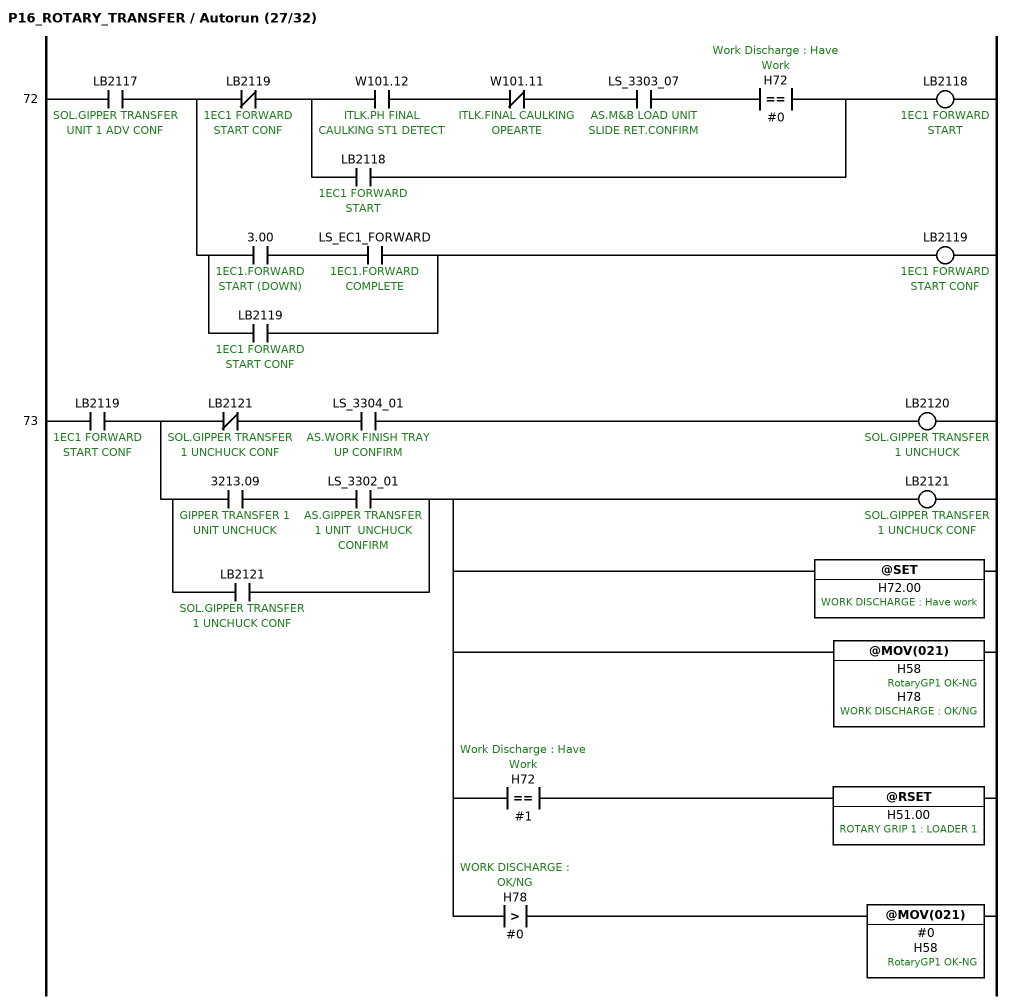
; [picture p264: P16_ROTARY_TRANSFER / Autorun, rungs 72-73]
; rung 72
LD LB2117  ; SOL.GIPPER TRANSFER UNIT 1 ADV CONF
OUT TR0
ANDNOT LB2119  ; 1EC1 FORWARD START CONF
LD W101.12  ; ITLK.PH FINAL CAULKING ST1 DETECT
ANDNOT W101.11  ; ITLK.FINAL CAULKING OPEARTE
AND LS_3303_07  ; AS.M&B LOAD UNIT SLIDE RET.CONFIRM
AND=(300) H72 #0  ; Work Discharge : Have Work
OR LB2118  ; 1EC1 FORWARD START
ANDLD
OUT LB2118  ; 1EC1 FORWARD START
LD TR0
LD 3.00  ; 1EC1.FORWARD START (DOWN)
AND LS_EC1_FORWARD  ; 1EC1.FORWARD COMPLETE
OR LB2119  ; 1EC1 FORWARD START CONF
ANDLD
OUT LB2119  ; 1EC1 FORWARD START CONF
; rung 73
LD LB2119  ; 1EC1 FORWARD START CONF
OUT TR0
ANDNOT LB2121  ; SOL.GIPPER TRANSFER 1 UNCHUCK CONF
AND LS_3304_01  ; AS.WORK FINISH TRAY UP CONFIRM
OUT LB2120  ; SOL.GIPPER TRANSFER 1 UNCHUCK
LD TR0
LD 3213.09  ; GIPPER TRANSFER 1 UNIT UNCHUCK
AND LS_3302_01  ; AS.GIPPER TRANSFER 1 UNIT  UNCHUCK CONFIRM
OR LB2121  ; SOL.GIPPER TRANSFER 1 UNCHUCK CONF
ANDLD
OUT TR0
OUT LB2121  ; SOL.GIPPER TRANSFER 1 UNCHUCK CONF
@SET H72.00  ; WORK DISCHARGE : Have work
@MOV(021) H58 H78  ; RotaryGP1 OK-NG, WORK DISCHARGE : OK/NG
AND=(300) H72 #1  ; Work Discharge : Have Work
@RSET H51.00  ; ROTARY GRIP 1 : LOADER 1
LD TR0
AND>(320) H78 #0  ; WORK DISCHARGE : OK/NG
@MOV(021) #0 H58  ; RotaryGP1 OK-NG

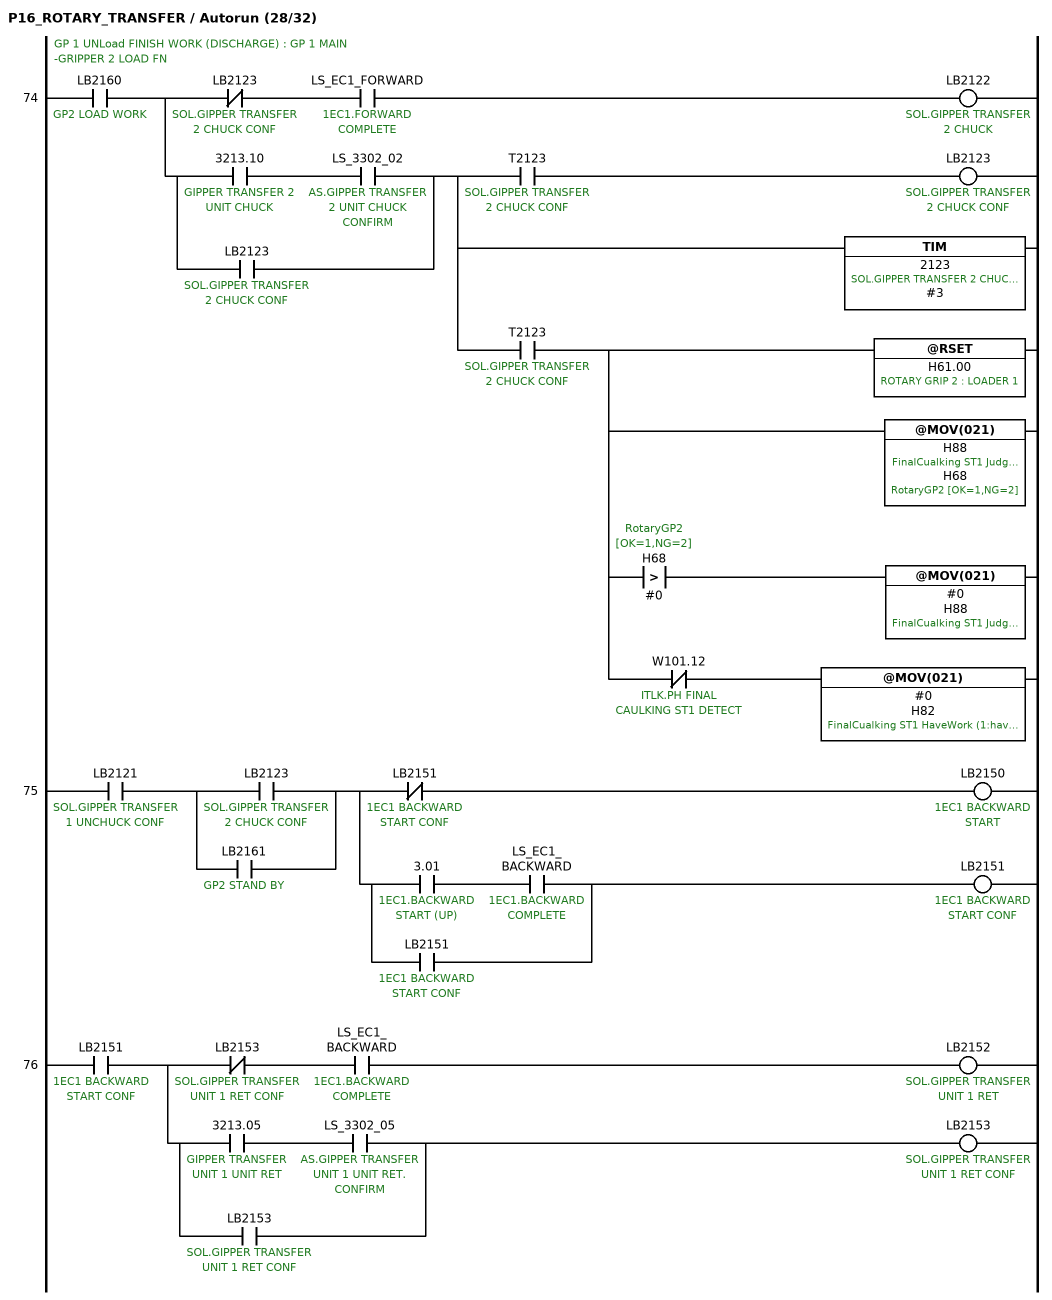
; rung 74: GP 1 UNLoad FINISH WORK (DISCHARGE) : GP 1 MAIN / -GRIPPER 2 LOAD FN
LD LB2160  ; GP2 LOAD WORK
OUT TR0
ANDNOT LB2123  ; SOL.GIPPER TRANSFER 2 CHUCK CONF
AND LS_EC1_FORWARD  ; 1EC1.FORWARD COMPLETE
OUT LB2122  ; SOL.GIPPER TRANSFER 2 CHUCK
LD TR0
LD 3213.10  ; GIPPER TRANSFER 2 UNIT CHUCK
AND LS_3302_02  ; AS.GIPPER TRANSFER 2 UNIT CHUCK CONFIRM
OR LB2123  ; SOL.GIPPER TRANSFER 2 CHUCK CONF
ANDLD
OUT TR0
AND T2123  ; SOL.GIPPER TRANSFER 2 CHUCK CONF
OUT LB2123  ; SOL.GIPPER TRANSFER 2 CHUCK CONF
LD TR0
TIM 2123 #3  ; SOL.GIPPER TRANSFER 2 CHUCK CONF
AND T2123  ; SOL.GIPPER TRANSFER 2 CHUCK CONF
OUT TR0
@RSET H61.00  ; ROTARY GRIP 2 : LOADER 1
@MOV(021) H88 H68  ; FinalCualking ST1 Judge [OK=1,NG=2], RotaryGP2 [OK=1,NG=2]
AND>(320) H68 #0  ; RotaryGP2 [OK=1,NG=2]
@MOV(021) #0 H88  ; FinalCualking ST1 Judge [OK=1,NG=2]
LD TR0
ANDNOT W101.12  ; ITLK.PH FINAL CAULKING ST1 DETECT
@MOV(021) #0 H82  ; FinalCualking ST1 HaveWork (1:have work 2:no work)
; rung 75
LD LB2121  ; SOL.GIPPER TRANSFER 1 UNCHUCK CONF
LD LB2123  ; SOL.GIPPER TRANSFER 2 CHUCK CONF
OR LB2161  ; GP2 STAND BY
ANDLD
OUT TR0
ANDNOT LB2151  ; 1EC1 BACKWARD START CONF
OUT LB2150  ; 1EC1 BACKWARD START
LD TR0
LD 3.01  ; 1EC1.BACKWARD START (UP)
AND LS_EC1_BACKWARD  ; 1EC1.BACKWARD COMPLETE
OR LB2151  ; 1EC1 BACKWARD START CONF
ANDLD
OUT LB2151  ; 1EC1 BACKWARD START CONF
; rung 76
LD LB2151  ; 1EC1 BACKWARD START CONF
OUT TR0
ANDNOT LB2153  ; SOL.GIPPER TRANSFER UNIT 1 RET CONF
AND LS_EC1_BACKWARD  ; 1EC1.BACKWARD COMPLETE
OUT LB2152  ; SOL.GIPPER TRANSFER UNIT 1 RET
LD TR0
LD 3213.05  ; GIPPER TRANSFER UNIT 1 UNIT RET
AND LS_3302_05  ; AS.GIPPER TRANSFER UNIT 1 UNIT RET. CONFIRM
OR LB2153  ; SOL.GIPPER TRANSFER UNIT 1 RET CONF
ANDLD
OUT LB2153  ; SOL.GIPPER TRANSFER UNIT 1 RET CONF

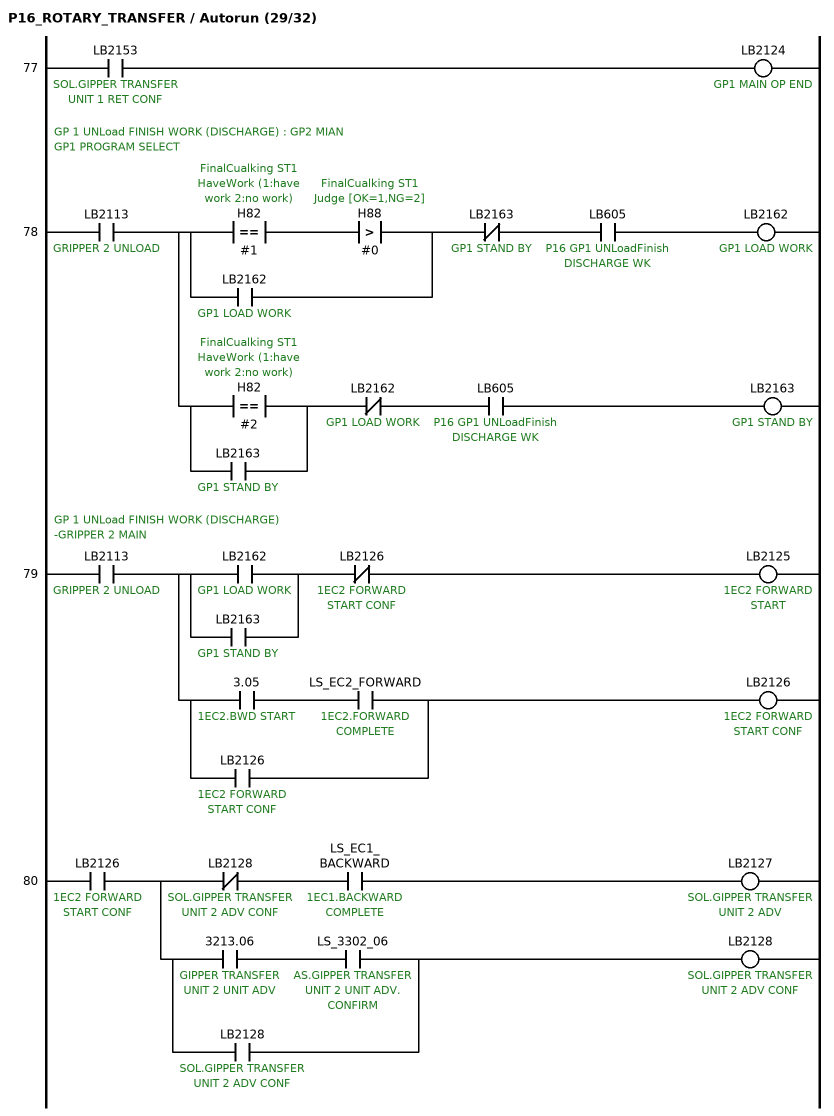
; rung 77
LD LB2153  ; SOL.GIPPER TRANSFER UNIT 1 RET CONF
OUT LB2124  ; GP1 MAIN OP END
; rung 78: GP 1 UNLoad FINISH WORK (DISCHARGE) : GP2 MIAN / GP1 PROGRAM SELECT
LD LB2113  ; GRIPPER 2 UNLOAD
OUT TR0
LD=(300) H82 #1  ; FinalCualking ST1 HaveWork (1:have work 2:no work)
AND>(320) H88 #0  ; FinalCualking ST1 Judge [OK=1,NG=2]
OR LB2162  ; GP1 LOAD WORK
ANDLD
ANDNOT LB2163  ; GP1 STAND BY
AND LB605  ; P16 GP1 UNLoadFinish DISCHARGE WK
OUT LB2162  ; GP1 LOAD WORK
LD TR0
LD=(300) H82 #2  ; FinalCualking ST1 HaveWork (1:have work 2:no work)
OR LB2163  ; GP1 STAND BY
ANDLD
ANDNOT LB2162  ; GP1 LOAD WORK
AND LB605  ; P16 GP1 UNLoadFinish DISCHARGE WK
OUT LB2163  ; GP1 STAND BY
; rung 79: GP 1 UNLoad FINISH WORK (DISCHARGE) / -GRIPPER 2 MAIN
LD LB2113  ; GRIPPER 2 UNLOAD
OUT TR0
LD LB2162  ; GP1 LOAD WORK
OR LB2163  ; GP1 STAND BY
ANDLD
ANDNOT LB2126  ; 1EC2 FORWARD START CONF
OUT LB2125  ; 1EC2 FORWARD START
LD TR0
LD 3.05  ; 1EC2.BWD START
AND LS_EC2_FORWARD  ; 1EC2.FORWARD COMPLETE
OR LB2126  ; 1EC2 FORWARD START CONF
ANDLD
OUT LB2126  ; 1EC2 FORWARD START CONF
; rung 80
LD LB2126  ; 1EC2 FORWARD START CONF
OUT TR0
ANDNOT LB2128  ; SOL.GIPPER TRANSFER UNIT 2 ADV CONF
AND LS_EC1_BACKWARD  ; 1EC1.BACKWARD COMPLETE
OUT LB2127  ; SOL.GIPPER TRANSFER UNIT 2 ADV
LD TR0
LD 3213.06  ; GIPPER TRANSFER UNIT 2 UNIT ADV
AND LS_3302_06  ; AS.GIPPER TRANSFER UNIT 2 UNIT ADV. CONFIRM
OR LB2128  ; SOL.GIPPER TRANSFER UNIT 2 ADV CONF
ANDLD
OUT LB2128  ; SOL.GIPPER TRANSFER UNIT 2 ADV CONF

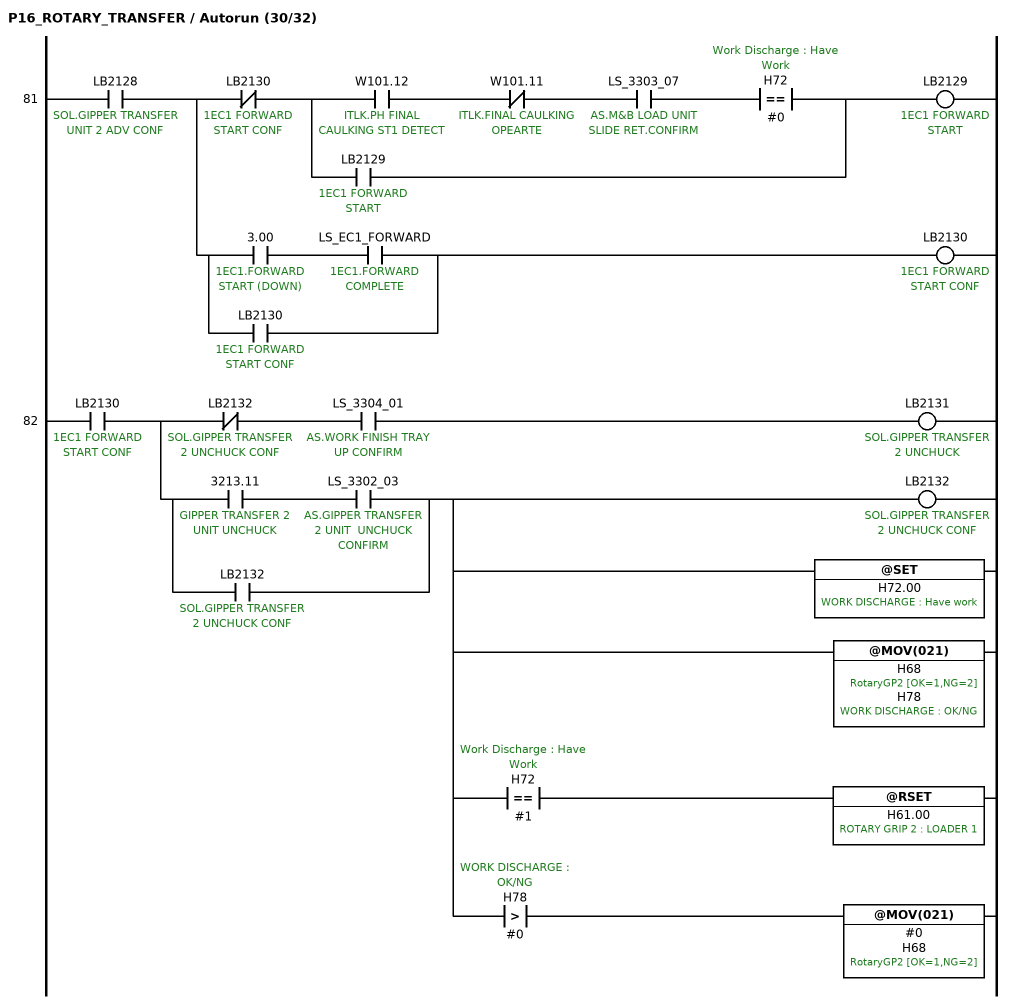
; rung 81
LD LB2128  ; SOL.GIPPER TRANSFER UNIT 2 ADV CONF
OUT TR0
ANDNOT LB2130  ; 1EC1 FORWARD START CONF
LD W101.12  ; ITLK.PH FINAL CAULKING ST1 DETECT
ANDNOT W101.11  ; ITLK.FINAL CAULKING OPEARTE
AND LS_3303_07  ; AS.M&B LOAD UNIT SLIDE RET.CONFIRM
AND=(300) H72 #0  ; Work Discharge : Have Work
OR LB2129  ; 1EC1 FORWARD START
ANDLD
OUT LB2129  ; 1EC1 FORWARD START
LD TR0
LD 3.00  ; 1EC1.FORWARD START (DOWN)
AND LS_EC1_FORWARD  ; 1EC1.FORWARD COMPLETE
OR LB2130  ; 1EC1 FORWARD START CONF
ANDLD
OUT LB2130  ; 1EC1 FORWARD START CONF
; rung 82
LD LB2130  ; 1EC1 FORWARD START CONF
OUT TR0
ANDNOT LB2132  ; SOL.GIPPER TRANSFER 2 UNCHUCK CONF
AND LS_3304_01  ; AS.WORK FINISH TRAY UP CONFIRM
OUT LB2131  ; SOL.GIPPER TRANSFER 2 UNCHUCK
LD TR0
LD 3213.11  ; GIPPER TRANSFER 2 UNIT UNCHUCK
AND LS_3302_03  ; AS.GIPPER TRANSFER 2 UNIT  UNCHUCK CONFIRM
OR LB2132  ; SOL.GIPPER TRANSFER 2 UNCHUCK CONF
ANDLD
OUT TR0
OUT LB2132  ; SOL.GIPPER TRANSFER 2 UNCHUCK CONF
@SET H72.00  ; WORK DISCHARGE : Have work
@MOV(021) H68 H78  ; RotaryGP2 [OK=1,NG=2], WORK DISCHARGE : OK/NG
AND=(300) H72 #1  ; Work Discharge : Have Work
@RSET H61.00  ; ROTARY GRIP 2 : LOADER 1
LD TR0
AND>(320) H78 #0  ; WORK DISCHARGE : OK/NG
@MOV(021) #0 H68  ; RotaryGP2 [OK=1,NG=2]

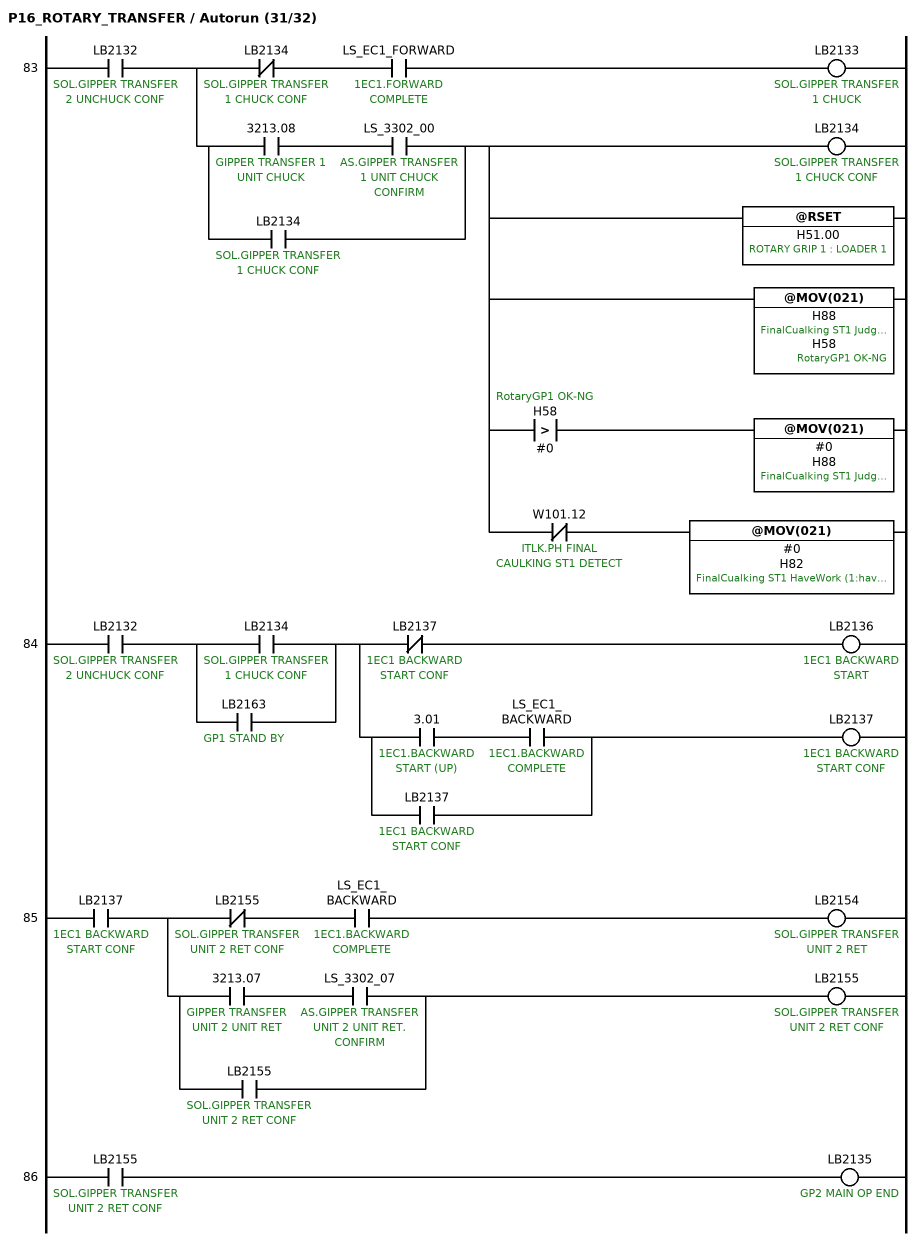
; rung 83
LD LB2132  ; SOL.GIPPER TRANSFER 2 UNCHUCK CONF
OUT TR0
ANDNOT LB2134  ; SOL.GIPPER TRANSFER 1 CHUCK CONF
AND LS_EC1_FORWARD  ; 1EC1.FORWARD COMPLETE
OUT LB2133  ; SOL.GIPPER TRANSFER 1 CHUCK
LD TR0
LD 3213.08  ; GIPPER TRANSFER 1 UNIT CHUCK
AND LS_3302_00  ; AS.GIPPER TRANSFER 1 UNIT CHUCK CONFIRM
OR LB2134  ; SOL.GIPPER TRANSFER 1 CHUCK CONF
ANDLD
OUT TR0
OUT LB2134  ; SOL.GIPPER TRANSFER 1 CHUCK CONF
@RSET H51.00  ; ROTARY GRIP 1 : LOADER 1
@MOV(021) H88 H58  ; FinalCualking ST1 Judge [OK=1,NG=2], RotaryGP1 OK-NG
AND>(320) H58 #0  ; RotaryGP1 OK-NG
@MOV(021) #0 H88  ; FinalCualking ST1 Judge [OK=1,NG=2]
LD TR0
ANDNOT W101.12  ; ITLK.PH FINAL CAULKING ST1 DETECT
@MOV(021) #0 H82  ; FinalCualking ST1 HaveWork (1:have work 2:no work)
; rung 84
LD LB2132  ; SOL.GIPPER TRANSFER 2 UNCHUCK CONF
LD LB2134  ; SOL.GIPPER TRANSFER 1 CHUCK CONF
OR LB2163  ; GP1 STAND BY
ANDLD
OUT TR0
ANDNOT LB2137  ; 1EC1 BACKWARD START CONF
OUT LB2136  ; 1EC1 BACKWARD START
LD TR0
LD 3.01  ; 1EC1.BACKWARD START (UP)
AND LS_EC1_BACKWARD  ; 1EC1.BACKWARD COMPLETE
OR LB2137  ; 1EC1 BACKWARD START CONF
ANDLD
OUT LB2137  ; 1EC1 BACKWARD START CONF
; rung 85
LD LB2137  ; 1EC1 BACKWARD START CONF
OUT TR0
ANDNOT LB2155  ; SOL.GIPPER TRANSFER UNIT 2 RET CONF
AND LS_EC1_BACKWARD  ; 1EC1.BACKWARD COMPLETE
OUT LB2154  ; SOL.GIPPER TRANSFER UNIT 2 RET
LD TR0
LD 3213.07  ; GIPPER TRANSFER UNIT 2 UNIT RET
AND LS_3302_07  ; AS.GIPPER TRANSFER UNIT 2 UNIT RET. CONFIRM
OR LB2155  ; SOL.GIPPER TRANSFER UNIT 2 RET CONF
ANDLD
OUT LB2155  ; SOL.GIPPER TRANSFER UNIT 2 RET CONF
; rung 86
LD LB2155  ; SOL.GIPPER TRANSFER UNIT 2 RET CONF
OUT LB2135  ; GP2 MAIN OP END

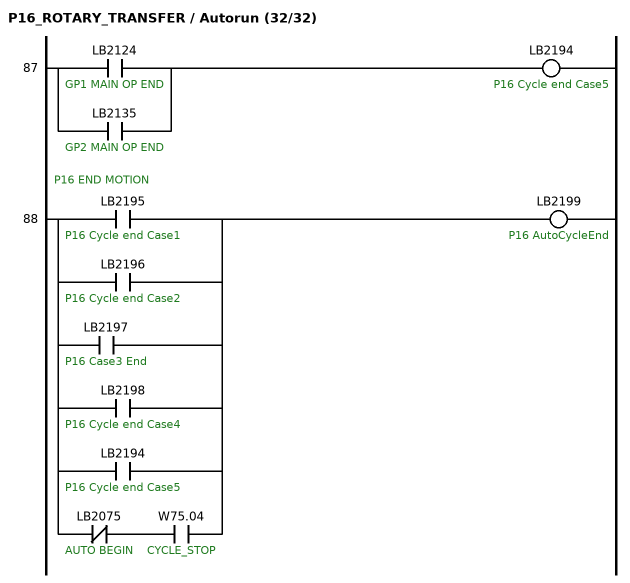
; rung 87
LD LB2124  ; GP1 MAIN OP END
OR LB2135  ; GP2 MAIN OP END
OUT LB2194  ; P16 Cycle end Case5
; rung 88: P16 END MOTION
LD LB2195  ; P16 Cycle end Case1
OR LB2196  ; P16 Cycle end Case2
OR LB2197  ; P16 Case3 End
OR LB2198  ; P16 Cycle end Case4
OR LB2194  ; P16 Cycle end Case5
LDNOT LB2075  ; AUTO BEGIN
AND W75.04  ; CYCLE_STOP
ORLD
OUT LB2199  ; P16 AutoCycleEnd

### Section Condition

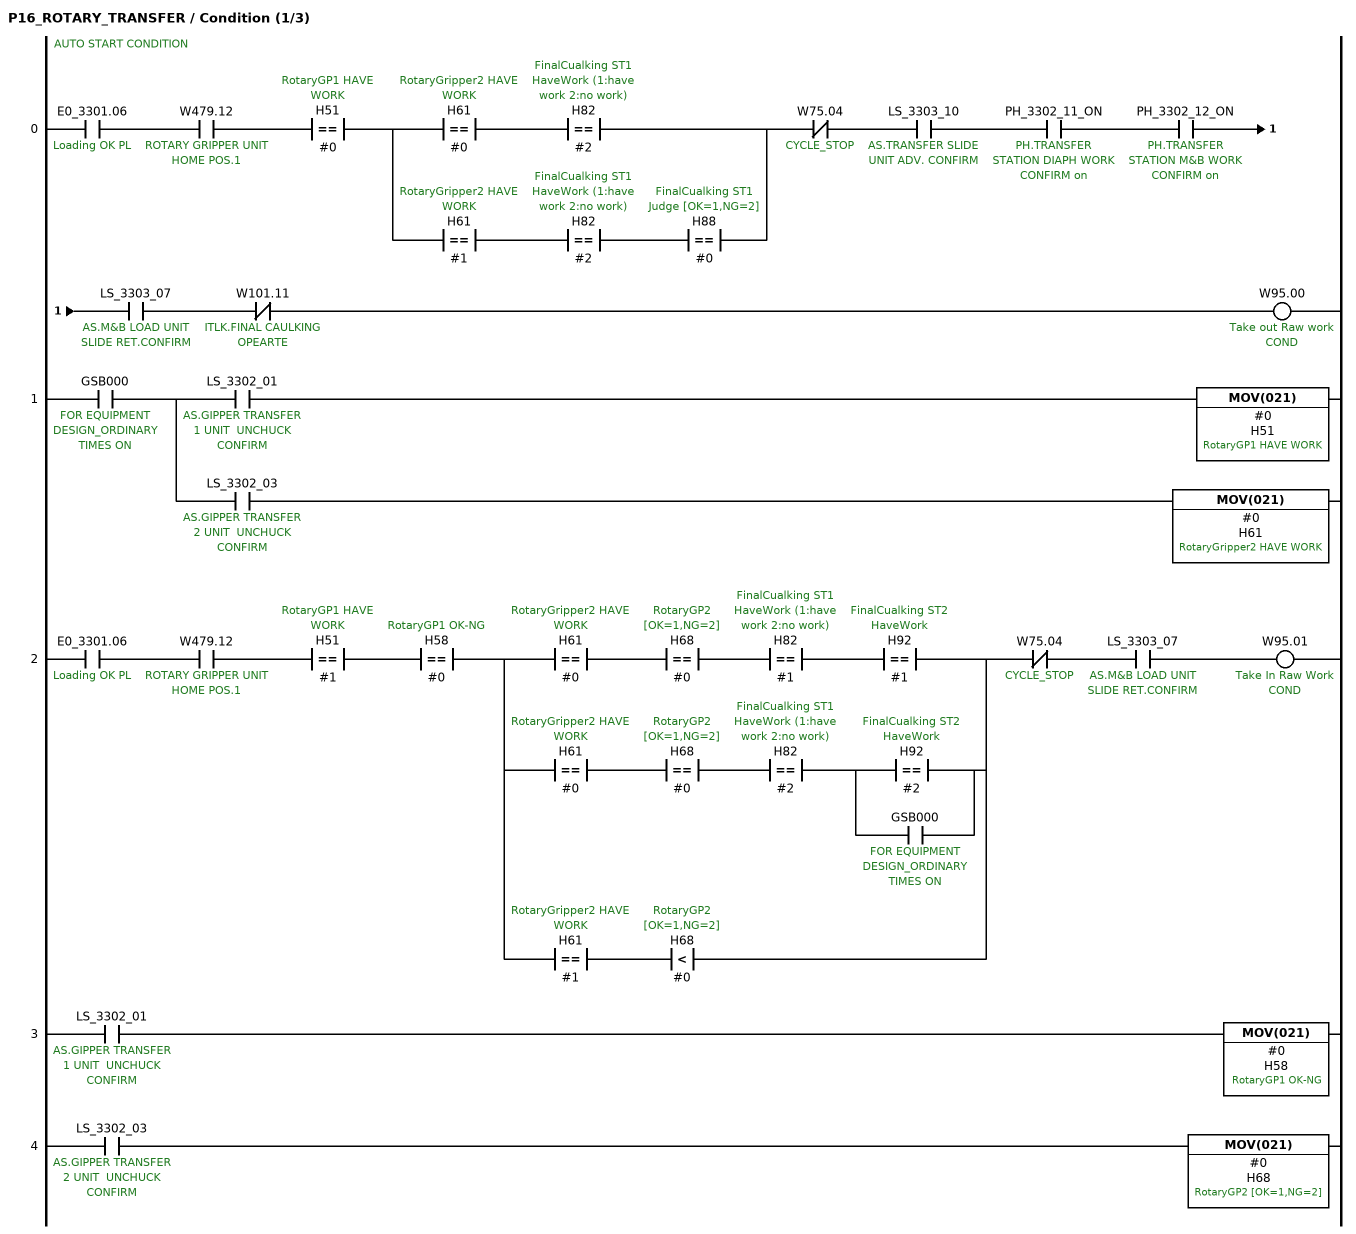
; rung 0: AUTO START CONDITION
LD E0_3301.06  ; Loading OK PL
AND W479.12  ; ROTARY GRIPPER UNIT HOME POS.1
AND=(300) H51 #0  ; RotaryGP1 HAVE WORK  // GP1 LOAD UNFINISH
LD=(300) H61 #0  ; RotaryGripper2 HAVE WORK  // GP2 STANDBY
AND=(300) H82 #2  ; FinalCualking ST1 HaveWork (1:have work 2:no work)
LD=(300) H61 #1  ; RotaryGripper2 HAVE WORK  // GP2 UNLOAD UNFINISH
AND=(300) H82 #2  ; FinalCualking ST1 HaveWork (1:have work 2:no work)
AND=(300) H88 #0  ; FinalCualking ST1 Judge [OK=1,NG=2]
ORLD
ANDLD
ANDNOT W75.04  ; CYCLE_STOP
AND LS_3303_10  ; AS.TRANSFER SLIDE UNIT ADV. CONFIRM
AND PH_3302_11_ON  ; PH.TRANSFER STATION DIAPH WORK CONFIRM on
AND PH_3302_12_ON  ; PH.TRANSFER STATION M&B WORK CONFIRM on
AND LS_3303_07  ; AS.M&B LOAD UNIT SLIDE RET.CONFIRM
ANDNOT W101.11  ; ITLK.FINAL CAULKING OPEARTE
OUT W95.00  ; Take out Raw work COND
; rung 1
LD GSB000  ; FOR EQUIPMENT DESIGN_ORDINARY TIMES ON
OUT TR0
AND LS_3302_01  ; AS.GIPPER TRANSFER 1 UNIT  UNCHUCK CONFIRM
MOV(021) #0 H51  ; RotaryGP1 HAVE WORK
LD TR0
AND LS_3302_03  ; AS.GIPPER TRANSFER 2 UNIT  UNCHUCK CONFIRM
MOV(021) #0 H61  ; RotaryGripper2 HAVE WORK
; rung 2
LD E0_3301.06  ; Loading OK PL
AND W479.12  ; ROTARY GRIPPER UNIT HOME POS.1
AND=(300) H51 #1  ; RotaryGP1 HAVE WORK  // GP1 UNLOAD UNFINISH
AND=(300) H58 #0  ; RotaryGP1 OK-NG
LD=(300) H61 #0  ; RotaryGripper2 HAVE WORK  // GP1&2 SPECIAL MOTION
AND=(300) H68 #0  ; RotaryGP2 [OK=1,NG=2]
AND=(300) H82 #1  ; FinalCualking ST1 HaveWork (1:have work 2:no work)
AND=(300) H92 #1  ; FinalCualking ST2 HaveWork
LD=(300) H61 #0  ; RotaryGripper2 HAVE WORK  // GP2 LOAD UNFINISH
AND=(300) H68 #0  ; RotaryGP2 [OK=1,NG=2]
AND=(300) H82 #2  ; FinalCualking ST1 HaveWork (1:have work 2:no work)
LD=(300) H92 #2  ; FinalCualking ST2 HaveWork
OR GSB000  ; FOR EQUIPMENT DESIGN_ORDINARY TIMES ON
ANDLD
ORLD
LD=(300) H61 #1  ; RotaryGripper2 HAVE WORK  // GP2 UNLOAD FINISH
AND<(310) H68 #0  ; RotaryGP2 [OK=1,NG=2]
ORLD
ANDLD
ANDNOT W75.04  ; CYCLE_STOP
AND LS_3303_07  ; AS.M&B LOAD UNIT SLIDE RET.CONFIRM
OUT W95.01  ; Take In Raw Work COND
; rung 3
LD LS_3302_01  ; AS.GIPPER TRANSFER 1 UNIT  UNCHUCK CONFIRM
MOV(021) #0 H58  ; RotaryGP1 OK-NG
; rung 4
LD LS_3302_03  ; AS.GIPPER TRANSFER 2 UNIT  UNCHUCK CONFIRM
MOV(021) #0 H68  ; RotaryGP2 [OK=1,NG=2]

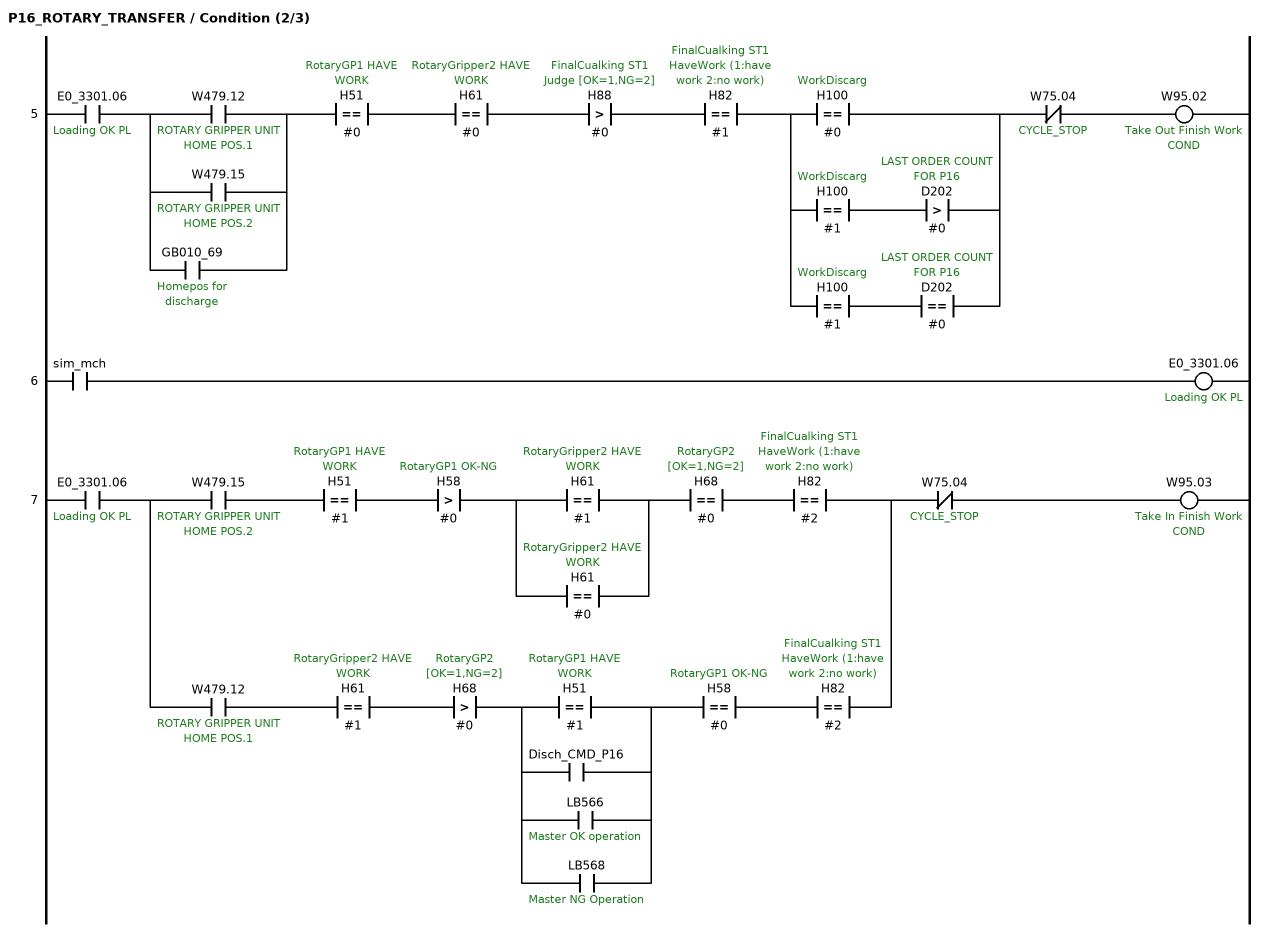
; rung 5
LD E0_3301.06  ; Loading OK PL
LD W479.12  ; ROTARY GRIPPER UNIT HOME POS.1
OR W479.15  ; ROTARY GRIPPER UNIT HOME POS.2
OR GB010_69  ; Homepos for discharge
ANDLD
AND=(300) H51 #0  ; RotaryGP1 HAVE WORK  // NORMAL HOME LOAD FINISH PALLAREL
AND=(300) H61 #0  ; RotaryGripper2 HAVE WORK
AND>(320) H88 #0  ; FinalCualking ST1 Judge [OK=1,NG=2]
AND=(300) H82 #1  ; FinalCualking ST1 HaveWork (1:have work 2:no work)
LD=(300) H100 #0  ; WorkDiscarg
LD=(300) H100 #1  ; WorkDiscarg  // GP1 LOAD FINISH TO DISCHARGE
AND>(320) D202 #0  ; LAST ORDER COUNT FOR P16
ORLD
LD=(300) H100 #1  ; WorkDiscarg  // GP1 LOAD FINISH TO DISCHARGE END
AND=(300) D202 #0  ; LAST ORDER COUNT FOR P16
ORLD
ANDLD
ANDNOT W75.04  ; CYCLE_STOP
OUT W95.02  ; Take Out Finish Work COND
; rung 6
LD sim_mch
OUT E0_3301.06  ; Loading OK PL
; rung 7
LD E0_3301.06  ; Loading OK PL
LD W479.15  ; ROTARY GRIPPER UNIT HOME POS.2
AND=(300) H51 #1  ; RotaryGP1 HAVE WORK  // MORMAL HOME UNLOAD FINISH
AND>(320) H58 #0  ; RotaryGP1 OK-NG
LD=(300) H61 #1  ; RotaryGripper2 HAVE WORK
OR=(300) H61 #0  ; RotaryGripper2 HAVE WORK
ANDLD
AND=(300) H68 #0  ; RotaryGP2 [OK=1,NG=2]
AND=(300) H82 #2  ; FinalCualking ST1 HaveWork (1:have work 2:no work)
LD W479.12  ; ROTARY GRIPPER UNIT HOME POS.1
AND=(300) H61 #1  ; RotaryGripper2 HAVE WORK  // REVERSE MORMAL HOME UNLOAD FINISH
AND>(320) H68 #0  ; RotaryGP2 [OK=1,NG=2]
LD=(300) H51 #1  ; RotaryGP1 HAVE WORK
OR Disch_CMD_P16
OR LB566  ; Master OK operation
OR LB568  ; Master NG Operation
ANDLD
AND=(300) H58 #0  ; RotaryGP1 OK-NG
AND=(300) H82 #2  ; FinalCualking ST1 HaveWork (1:have work 2:no work)
ORLD
ANDLD
ANDNOT W75.04  ; CYCLE_STOP
OUT W95.03  ; Take In Finish Work COND

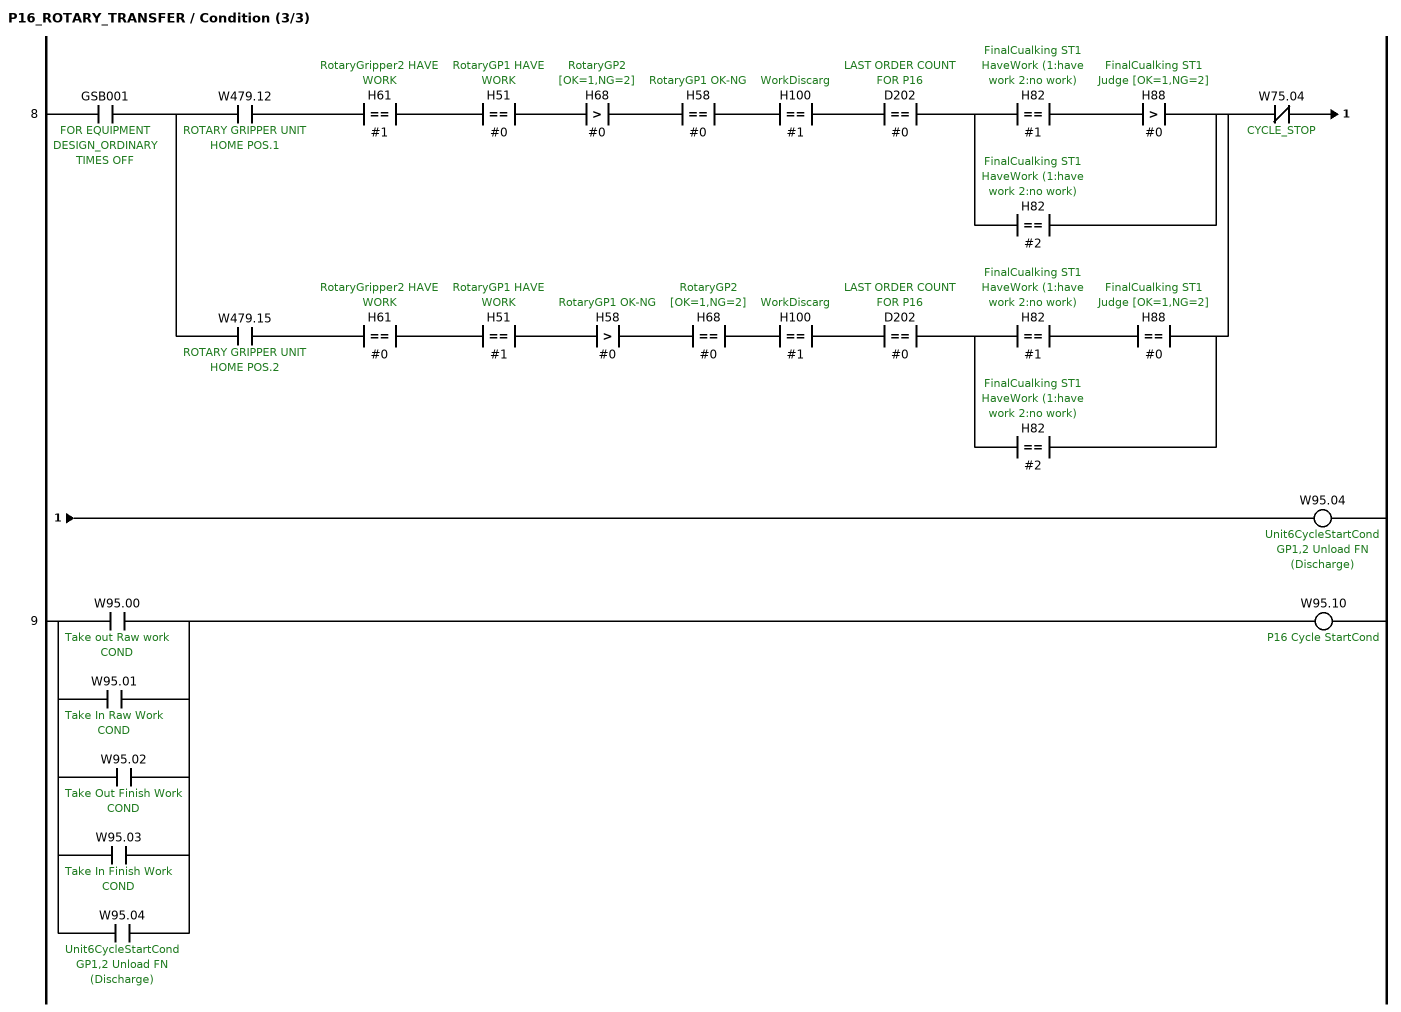
; rung 8
LD GSB001  ; FOR EQUIPMENT DESIGN_ORDINARY TIMES OFF
LD W479.12  ; ROTARY GRIPPER UNIT HOME POS.1
AND=(300) H61 #1  ; RotaryGripper2 HAVE WORK
AND=(300) H51 #0  ; RotaryGP1 HAVE WORK
AND>(320) H68 #0  ; RotaryGP2 [OK=1,NG=2]
AND=(300) H58 #0  ; RotaryGP1 OK-NG
AND=(300) H100 #1  ; WorkDiscarg
AND=(300) D202 #0  ; LAST ORDER COUNT FOR P16
LD=(300) H82 #1  ; FinalCualking ST1 HaveWork (1:have work 2:no work)
AND>(320) H88 #0  ; FinalCualking ST1 Judge [OK=1,NG=2]
OR=(300) H82 #2  ; FinalCualking ST1 HaveWork (1:have work 2:no work)
ANDLD
LD W479.15  ; ROTARY GRIPPER UNIT HOME POS.2
AND=(300) H61 #0  ; RotaryGripper2 HAVE WORK
AND=(300) H51 #1  ; RotaryGP1 HAVE WORK
AND>(320) H58 #0  ; RotaryGP1 OK-NG
AND=(300) H68 #0  ; RotaryGP2 [OK=1,NG=2]
AND=(300) H100 #1  ; WorkDiscarg
AND=(300) D202 #0  ; LAST ORDER COUNT FOR P16
LD=(300) H82 #1  ; FinalCualking ST1 HaveWork (1:have work 2:no work)
AND=(300) H88 #0  ; FinalCualking ST1 Judge [OK=1,NG=2]
OR=(300) H82 #2  ; FinalCualking ST1 HaveWork (1:have work 2:no work)
ANDLD
ORLD
ANDLD
ANDNOT W75.04  ; CYCLE_STOP
OUT W95.04  ; Unit6CycleStartCond GP1,2 Unload FN (Discharge)
; rung 9
LD W95.00  ; Take out Raw work COND
OR W95.01  ; Take In Raw Work COND
OR W95.02  ; Take Out Finish Work COND
OR W95.03  ; Take In Finish Work COND
OR W95.04  ; Unit6CycleStartCond GP1,2 Unload FN (Discharge)
OUT W95.10  ; P16 Cycle StartCond

### Section Device_Output

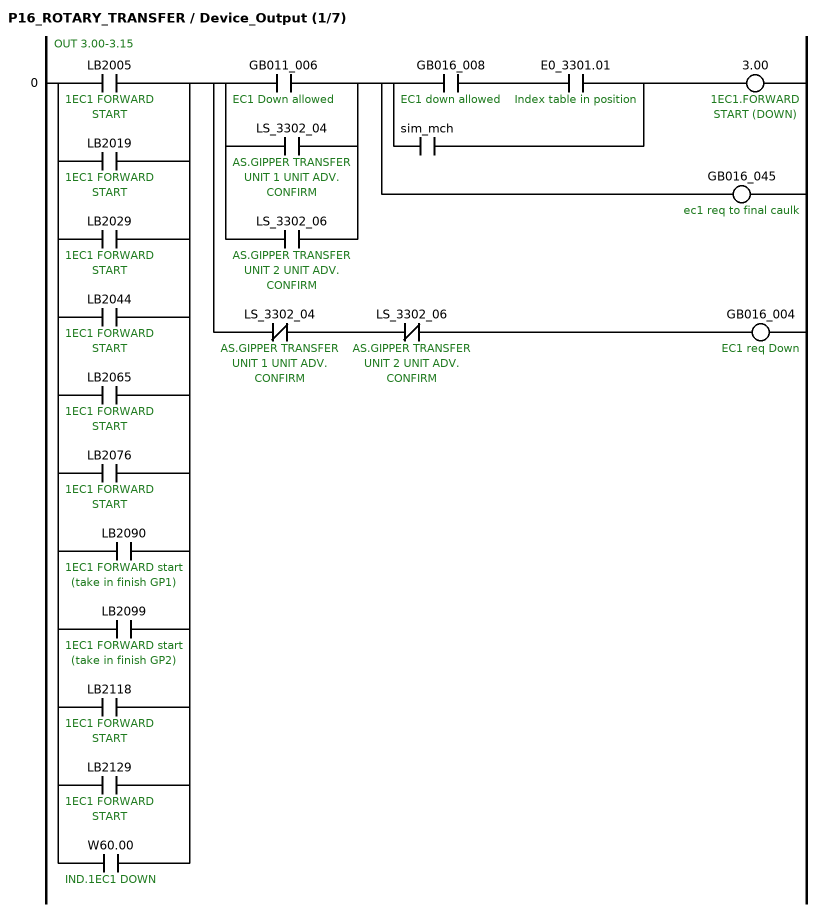
; rung 0: OUT 3.00-3.15
LD LB2005  ; 1EC1 FORWARD START
OR LB2019  ; 1EC1 FORWARD START
OR LB2029  ; 1EC1 FORWARD START
OR LB2044  ; 1EC1 FORWARD START
OR LB2065  ; 1EC1 FORWARD START
OR LB2076  ; 1EC1 FORWARD START
OR LB2090  ; 1EC1 FORWARD start (take in finish GP1)
OR LB2099  ; 1EC1 FORWARD start (take in finish GP2)
OR LB2118  ; 1EC1 FORWARD START
OR LB2129  ; 1EC1 FORWARD START
OR W60.00  ; IND.1EC1 DOWN
OUT TR0
LD GB011_006  ; EC1 Down allowed
OR LS_3302_04  ; AS.GIPPER TRANSFER UNIT 1 UNIT ADV. CONFIRM
OR LS_3302_06  ; AS.GIPPER TRANSFER UNIT 2 UNIT ADV. CONFIRM
ANDLD
OUT TR1
LD GB016_008  ; EC1 down allowed
AND E0_3301.01  ; Index table in position
OR sim_mch
ANDLD
OUT 3.00  ; 1EC1.FORWARD START (DOWN)
LD TR1
OUT GB016_045  ; ec1 req to final caulk
LD TR0
ANDNOT LS_3302_04  ; AS.GIPPER TRANSFER UNIT 1 UNIT ADV. CONFIRM
ANDNOT LS_3302_06  ; AS.GIPPER TRANSFER UNIT 2 UNIT ADV. CONFIRM
OUT GB016_004  ; EC1 req Down

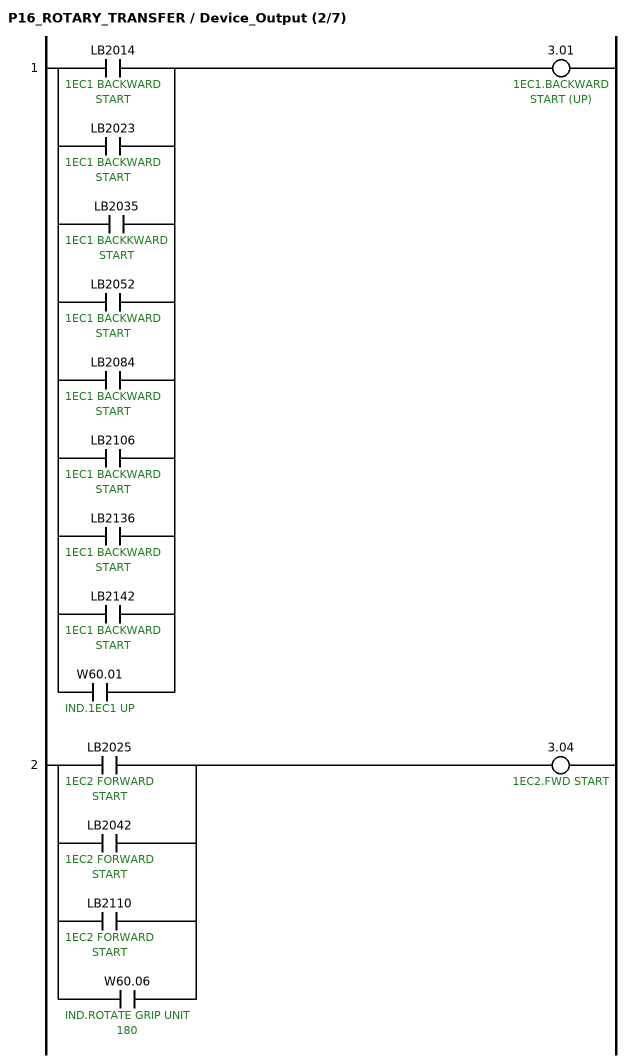
; rung 1
LD LB2014  ; 1EC1 BACKWARD START
OR LB2023  ; 1EC1 BACKWARD START
OR LB2035  ; 1EC1 BACKKWARD START
OR LB2052  ; 1EC1 BACKWARD START
OR LB2084  ; 1EC1 BACKWARD START
OR LB2106  ; 1EC1 BACKWARD START
OR LB2136  ; 1EC1 BACKWARD START
OR LB2142  ; 1EC1 BACKWARD START
OR W60.01  ; IND.1EC1 UP
OUT 3.01  ; 1EC1.BACKWARD START (UP)
; rung 2
LD LB2025  ; 1EC2 FORWARD START
OR LB2042  ; 1EC2 FORWARD START
OR LB2110  ; 1EC2 FORWARD START
OR W60.06  ; IND.ROTATE GRIP UNIT 180
OUT 3.04  ; 1EC2.FWD START

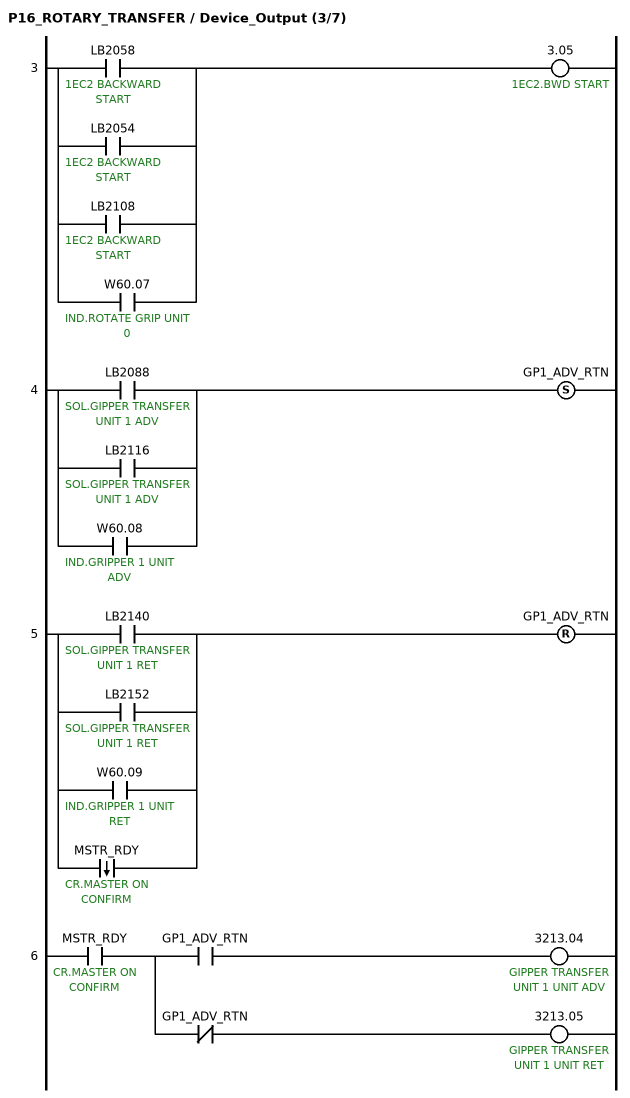
; rung 3
LD LB2058  ; 1EC2 BACKWARD START
OR LB2054  ; 1EC2 BACKWARD START
OR LB2108  ; 1EC2 BACKWARD START
OR W60.07  ; IND.ROTATE GRIP UNIT 0
OUT 3.05  ; 1EC2.BWD START
; rung 4
LD LB2088  ; SOL.GIPPER TRANSFER UNIT 1 ADV
OR LB2116  ; SOL.GIPPER TRANSFER UNIT 1 ADV
OR W60.08  ; IND.GRIPPER 1 UNIT ADV
SET GP1_ADV_RTN
; rung 5
LD LB2140  ; SOL.GIPPER TRANSFER UNIT 1 RET
OR LB2152  ; SOL.GIPPER TRANSFER UNIT 1 RET
OR W60.09  ; IND.GRIPPER 1 UNIT RET
%OR MSTR_RDY  ; CR.MASTER ON CONFIRM
RSET GP1_ADV_RTN
; rung 6
LD MSTR_RDY  ; CR.MASTER ON CONFIRM
OUT TR0
AND GP1_ADV_RTN
OUT 3213.04  ; GIPPER TRANSFER UNIT 1 UNIT ADV
LD TR0
ANDNOT GP1_ADV_RTN
OUT 3213.05  ; GIPPER TRANSFER UNIT 1 UNIT RET

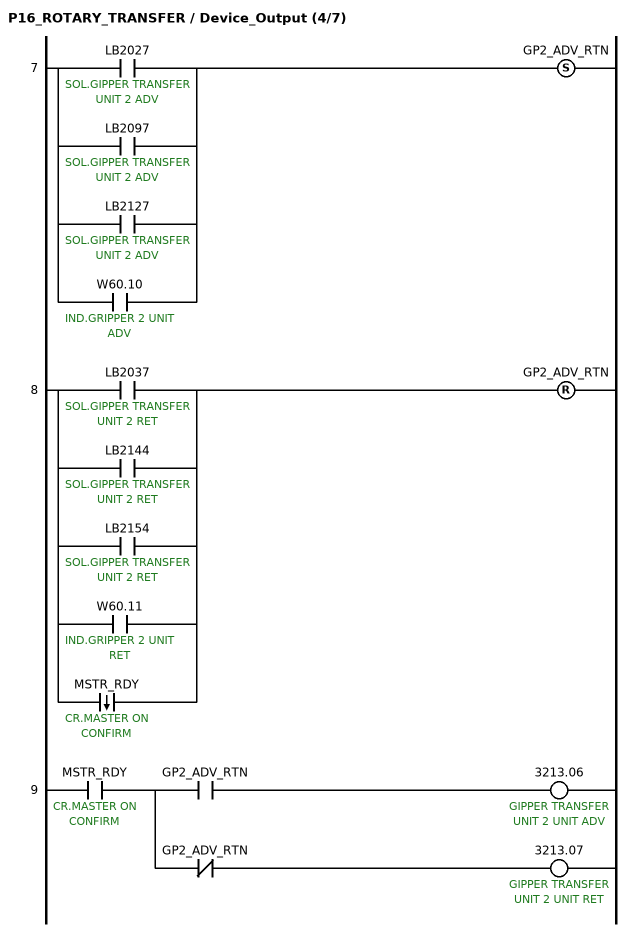
; rung 7
LD LB2027  ; SOL.GIPPER TRANSFER UNIT 2 ADV
OR LB2097  ; SOL.GIPPER TRANSFER UNIT 2 ADV
OR LB2127  ; SOL.GIPPER TRANSFER UNIT 2 ADV
OR W60.10  ; IND.GRIPPER 2 UNIT ADV
SET GP2_ADV_RTN
; rung 8
LD LB2037  ; SOL.GIPPER TRANSFER UNIT 2 RET
OR LB2144  ; SOL.GIPPER TRANSFER UNIT 2 RET
OR LB2154  ; SOL.GIPPER TRANSFER UNIT 2 RET
OR W60.11  ; IND.GRIPPER 2 UNIT RET
%OR MSTR_RDY  ; CR.MASTER ON CONFIRM
RSET GP2_ADV_RTN
; rung 9
LD MSTR_RDY  ; CR.MASTER ON CONFIRM
OUT TR0
AND GP2_ADV_RTN
OUT 3213.06  ; GIPPER TRANSFER UNIT 2 UNIT ADV
LD TR0
ANDNOT GP2_ADV_RTN
OUT 3213.07  ; GIPPER TRANSFER UNIT 2 UNIT RET

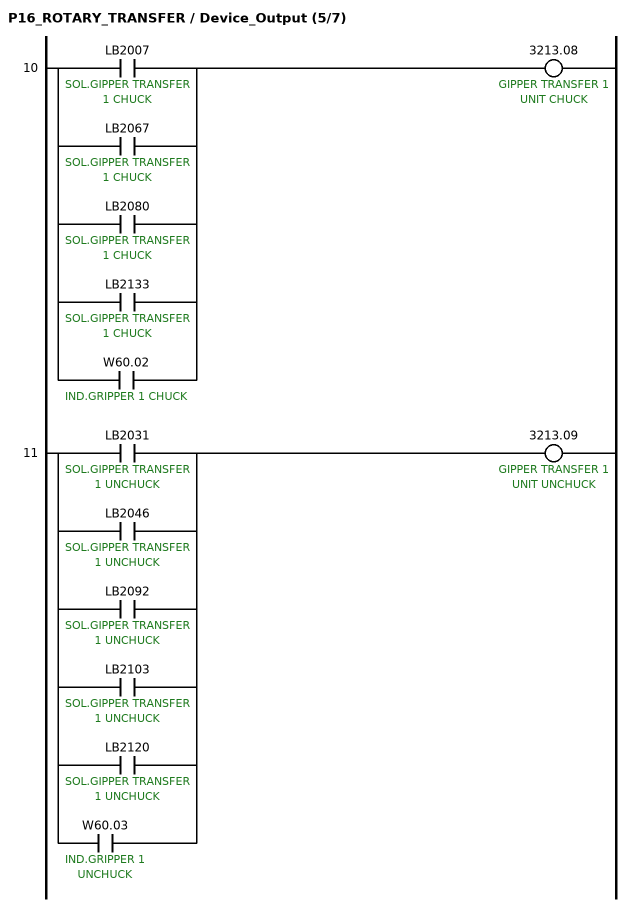
; rung 10
LD LB2007  ; SOL.GIPPER TRANSFER 1 CHUCK
OR LB2067  ; SOL.GIPPER TRANSFER 1 CHUCK
OR LB2080  ; SOL.GIPPER TRANSFER 1 CHUCK
OR LB2133  ; SOL.GIPPER TRANSFER 1 CHUCK
OR W60.02  ; IND.GRIPPER 1 CHUCK
OUT 3213.08  ; GIPPER TRANSFER 1 UNIT CHUCK
; rung 11
LD LB2031  ; SOL.GIPPER TRANSFER 1 UNCHUCK
OR LB2046  ; SOL.GIPPER TRANSFER 1 UNCHUCK
OR LB2092  ; SOL.GIPPER TRANSFER 1 UNCHUCK
OR LB2103  ; SOL.GIPPER TRANSFER 1 UNCHUCK
OR LB2120  ; SOL.GIPPER TRANSFER 1 UNCHUCK
OR W60.03  ; IND.GRIPPER 1 UNCHUCK
OUT 3213.09  ; GIPPER TRANSFER 1 UNIT UNCHUCK

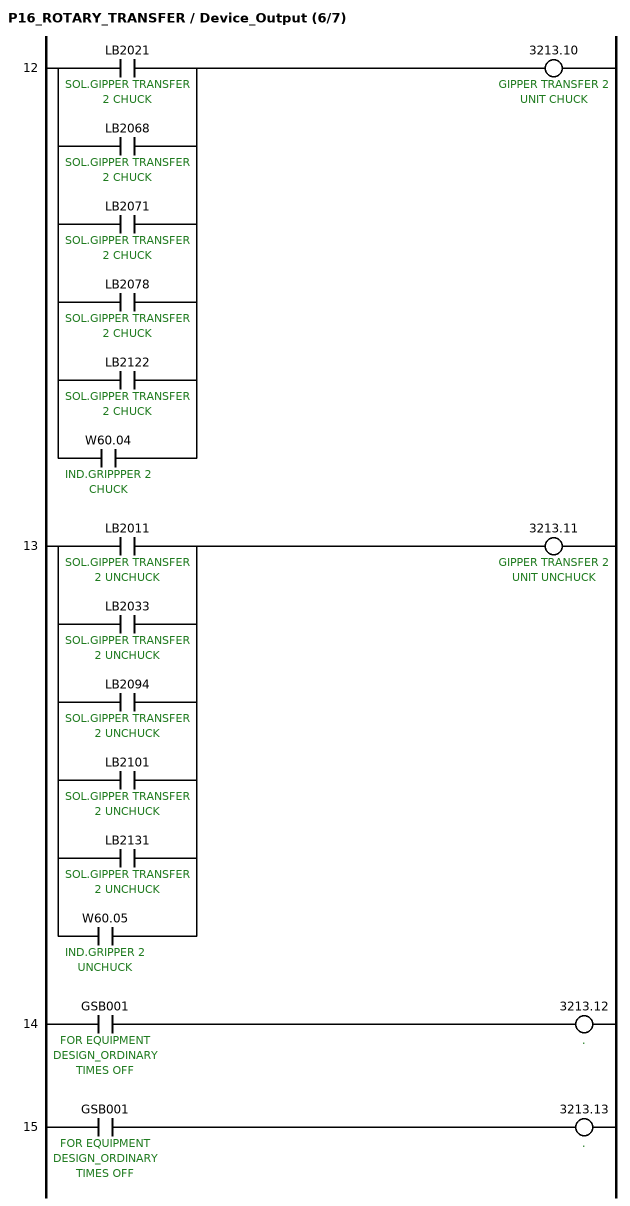
; rung 12
LD LB2021  ; SOL.GIPPER TRANSFER 2 CHUCK
OR LB2068  ; SOL.GIPPER TRANSFER 2 CHUCK
OR LB2071  ; SOL.GIPPER TRANSFER 2 CHUCK
OR LB2078  ; SOL.GIPPER TRANSFER 2 CHUCK
OR LB2122  ; SOL.GIPPER TRANSFER 2 CHUCK
OR W60.04  ; IND.GRIPPPER 2 CHUCK
OUT 3213.10  ; GIPPER TRANSFER 2 UNIT CHUCK
; rung 13
LD LB2011  ; SOL.GIPPER TRANSFER 2 UNCHUCK
OR LB2033  ; SOL.GIPPER TRANSFER 2 UNCHUCK
OR LB2094  ; SOL.GIPPER TRANSFER 2 UNCHUCK
OR LB2101  ; SOL.GIPPER TRANSFER 2 UNCHUCK
OR LB2131  ; SOL.GIPPER TRANSFER 2 UNCHUCK
OR W60.05  ; IND.GRIPPER 2 UNCHUCK
OUT 3213.11  ; GIPPER TRANSFER 2 UNIT UNCHUCK
; rung 14
LD GSB001  ; FOR EQUIPMENT DESIGN_ORDINARY TIMES OFF
OUT 3213.12  ; .
; rung 15
LD GSB001  ; FOR EQUIPMENT DESIGN_ORDINARY TIMES OFF
OUT 3213.13  ; .

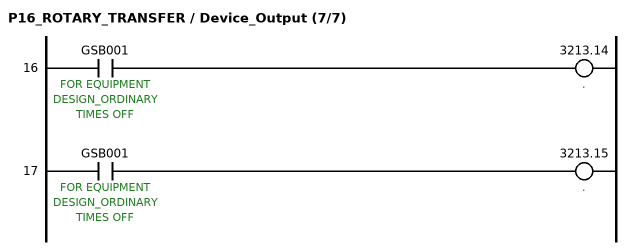
; rung 16
LD GSB001  ; FOR EQUIPMENT DESIGN_ORDINARY TIMES OFF
OUT 3213.14  ; .
; rung 17
LD GSB001  ; FOR EQUIPMENT DESIGN_ORDINARY TIMES OFF
OUT 3213.15  ; .

### Section Station_Output

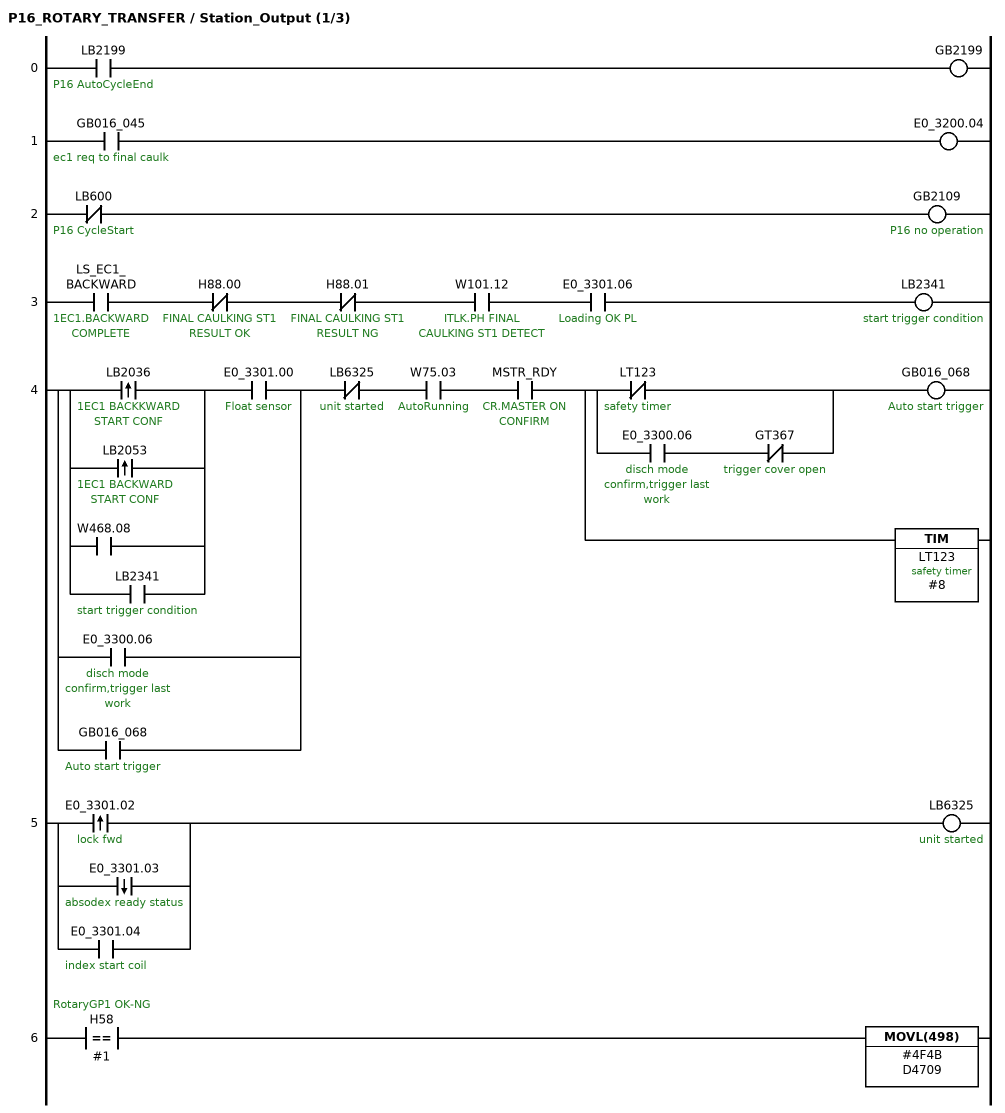
; rung 0
LD LB2199  ; P16 AutoCycleEnd
OUT GB2199
; rung 1
LD GB016_045  ; ec1 req to final caulk
OUT E0_3200.04
; rung 2
LDNOT LB600  ; P16 CycleStart
OUT GB2109  ; P16 no operation
; rung 3
LD LS_EC1_BACKWARD  ; 1EC1.BACKWARD COMPLETE
ANDNOT H88.00  ; FINAL CAULKING ST1 RESULT OK
ANDNOT H88.01  ; FINAL CAULKING ST1 RESULT NG
AND W101.12  ; ITLK.PH FINAL CAULKING ST1 DETECT
AND E0_3301.06  ; Loading OK PL
OUT LB2341  ; start trigger condition
; rung 4
@LD LB2036  ; 1EC1 BACKKWARD START CONF
@OR LB2053  ; 1EC1 BACKWARD START CONF
OR W468.08
OR LB2341  ; start trigger condition
AND E0_3301.00  ; Float sensor
OR E0_3300.06  ; disch mode confirm,trigger last work
OR GB016_068  ; Auto start trigger
ANDNOT LB6325  ; unit started
AND W75.03  ; AutoRunning
AND MSTR_RDY  ; CR.MASTER ON CONFIRM
OUT TR0
LDNOT LT123  ; safety timer
LD E0_3300.06  ; disch mode confirm,trigger last work
ANDNOT GT367  ; trigger cover open
ORLD
ANDLD
OUT GB016_068  ; Auto start trigger
LD TR0
TIM LT123 #8  ; safety timer
; rung 5
@LD E0_3301.02  ; lock fwd
%OR E0_3301.03  ; absodex ready status
OR E0_3301.04  ; index start coil
OUT LB6325  ; unit started
; rung 6
LD=(300) H58 #1  ; RotaryGP1 OK-NG
MOVL(498) #4F4B D4709

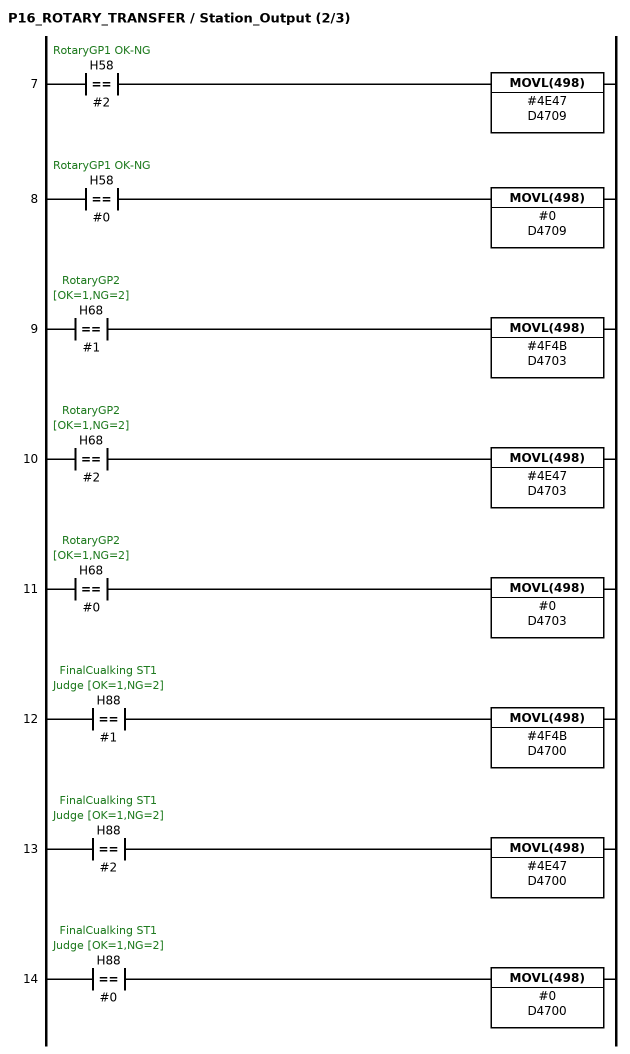
; rung 7
LD=(300) H58 #2  ; RotaryGP1 OK-NG
MOVL(498) #4E47 D4709
; rung 8
LD=(300) H58 #0  ; RotaryGP1 OK-NG
MOVL(498) #0 D4709
; rung 9
LD=(300) H68 #1  ; RotaryGP2 [OK=1,NG=2]
MOVL(498) #4F4B D4703
; rung 10
LD=(300) H68 #2  ; RotaryGP2 [OK=1,NG=2]
MOVL(498) #4E47 D4703
; rung 11
LD=(300) H68 #0  ; RotaryGP2 [OK=1,NG=2]
MOVL(498) #0 D4703
; rung 12
LD=(300) H88 #1  ; FinalCualking ST1 Judge [OK=1,NG=2]
MOVL(498) #4F4B D4700
; rung 13
LD=(300) H88 #2  ; FinalCualking ST1 Judge [OK=1,NG=2]
MOVL(498) #4E47 D4700
; rung 14
LD=(300) H88 #0  ; FinalCualking ST1 Judge [OK=1,NG=2]
MOVL(498) #0 D4700

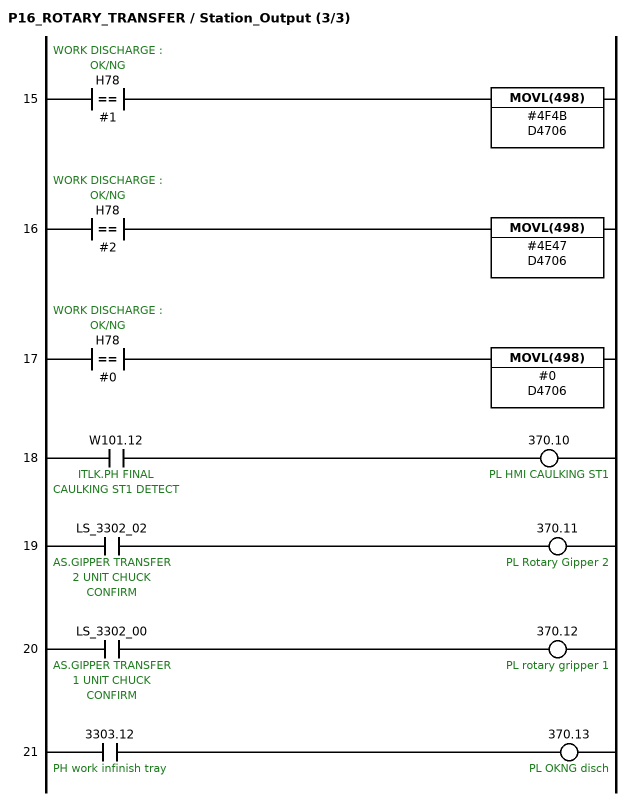
; rung 15
LD=(300) H78 #1  ; WORK DISCHARGE : OK/NG
MOVL(498) #4F4B D4706
; rung 16
LD=(300) H78 #2  ; WORK DISCHARGE : OK/NG
MOVL(498) #4E47 D4706
; rung 17
LD=(300) H78 #0  ; WORK DISCHARGE : OK/NG
MOVL(498) #0 D4706
; rung 18
LD W101.12  ; ITLK.PH FINAL CAULKING ST1 DETECT
OUT 370.10  ; PL HMI CAULKING ST1
; rung 19
LD LS_3302_02  ; AS.GIPPER TRANSFER 2 UNIT CHUCK CONFIRM
OUT 370.11  ; PL Rotary Gipper 2
; rung 20
LD LS_3302_00  ; AS.GIPPER TRANSFER 1 UNIT CHUCK CONFIRM
OUT 370.12  ; PL rotary gripper 1
; rung 21
LD 3303.12  ; PH work infinish tray
OUT 370.13  ; PL OKNG disch

### Section Individual

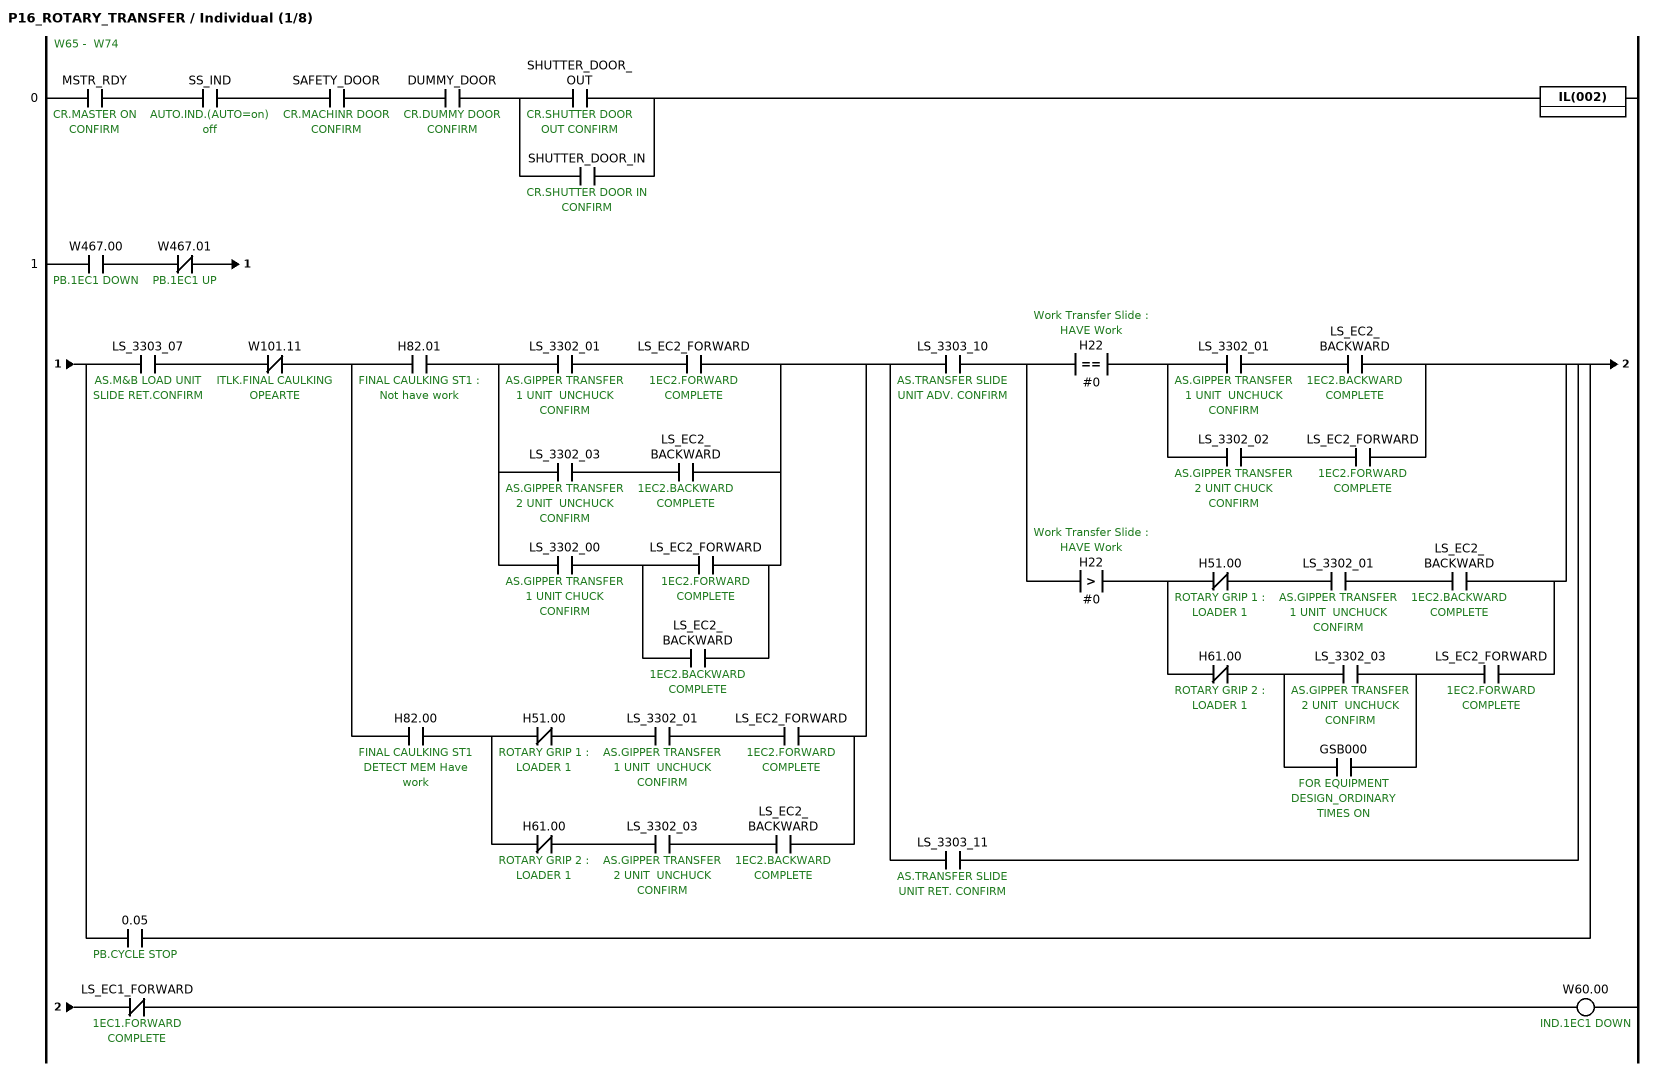
; rung 0: W65 -  W74
LD MSTR_RDY  ; CR.MASTER ON CONFIRM
AND SS_IND  ; AUTO.IND.(AUTO=on) off
AND SAFETY_DOOR  ; CR.MACHINR DOOR CONFIRM
AND DUMMY_DOOR  ; CR.DUMMY DOOR CONFIRM
LD SHUTTER_DOOR_OUT  ; CR.SHUTTER DOOR OUT CONFIRM
OR SHUTTER_DOOR_IN  ; CR.SHUTTER DOOR IN CONFIRM
ANDLD
IL(002)
; rung 1
LD W467.00  ; PB.1EC1 DOWN
ANDNOT W467.01  ; PB.1EC1 UP
LD LS_3303_07  ; AS.M&B LOAD UNIT SLIDE RET.CONFIRM
ANDNOT W101.11  ; ITLK.FINAL CAULKING OPEARTE
LD H82.01  ; FINAL CAULKING ST1 : Not have work
LD LS_3302_01  ; AS.GIPPER TRANSFER 1 UNIT  UNCHUCK CONFIRM
AND LS_EC2_FORWARD  ; 1EC2.FORWARD COMPLETE
LD LS_3302_03  ; AS.GIPPER TRANSFER 2 UNIT  UNCHUCK CONFIRM
AND LS_EC2_BACKWARD  ; 1EC2.BACKWARD COMPLETE
ORLD
LD LS_3302_00  ; AS.GIPPER TRANSFER 1 UNIT CHUCK CONFIRM
LD LS_EC2_FORWARD  ; 1EC2.FORWARD COMPLETE
OR LS_EC2_BACKWARD  ; 1EC2.BACKWARD COMPLETE
ANDLD
ORLD
ANDLD
LD H82.00  ; FINAL CAULKING ST1 DETECT MEM Have work
LDNOT H51.00  ; ROTARY GRIP 1 : LOADER 1
AND LS_3302_01  ; AS.GIPPER TRANSFER 1 UNIT  UNCHUCK CONFIRM
AND LS_EC2_FORWARD  ; 1EC2.FORWARD COMPLETE
LDNOT H61.00  ; ROTARY GRIP 2 : LOADER 1
AND LS_3302_03  ; AS.GIPPER TRANSFER 2 UNIT  UNCHUCK CONFIRM
AND LS_EC2_BACKWARD  ; 1EC2.BACKWARD COMPLETE
ORLD
ANDLD
ORLD
ANDLD
LD LS_3303_10  ; AS.TRANSFER SLIDE UNIT ADV. CONFIRM
LD=(300) H22 #0  ; Work Transfer Slide : HAVE Work
LD LS_3302_01  ; AS.GIPPER TRANSFER 1 UNIT  UNCHUCK CONFIRM
AND LS_EC2_BACKWARD  ; 1EC2.BACKWARD COMPLETE
LD LS_3302_02  ; AS.GIPPER TRANSFER 2 UNIT CHUCK CONFIRM
AND LS_EC2_FORWARD  ; 1EC2.FORWARD COMPLETE
ORLD
ANDLD
LD>(320) H22 #0  ; Work Transfer Slide : HAVE Work
LDNOT H51.00  ; ROTARY GRIP 1 : LOADER 1
AND LS_3302_01  ; AS.GIPPER TRANSFER 1 UNIT  UNCHUCK CONFIRM
AND LS_EC2_BACKWARD  ; 1EC2.BACKWARD COMPLETE
LDNOT H61.00  ; ROTARY GRIP 2 : LOADER 1
LD LS_3302_03  ; AS.GIPPER TRANSFER 2 UNIT  UNCHUCK CONFIRM
OR GSB000  ; FOR EQUIPMENT DESIGN_ORDINARY TIMES ON
ANDLD
AND LS_EC2_FORWARD  ; 1EC2.FORWARD COMPLETE
ORLD
ANDLD
ORLD
ANDLD
OR LS_3303_11  ; AS.TRANSFER SLIDE UNIT RET. CONFIRM
ANDLD
OR 0.05  ; PB.CYCLE STOP
ANDLD
ANDNOT LS_EC1_FORWARD  ; 1EC1.FORWARD COMPLETE
OUT W60.00  ; IND.1EC1 DOWN

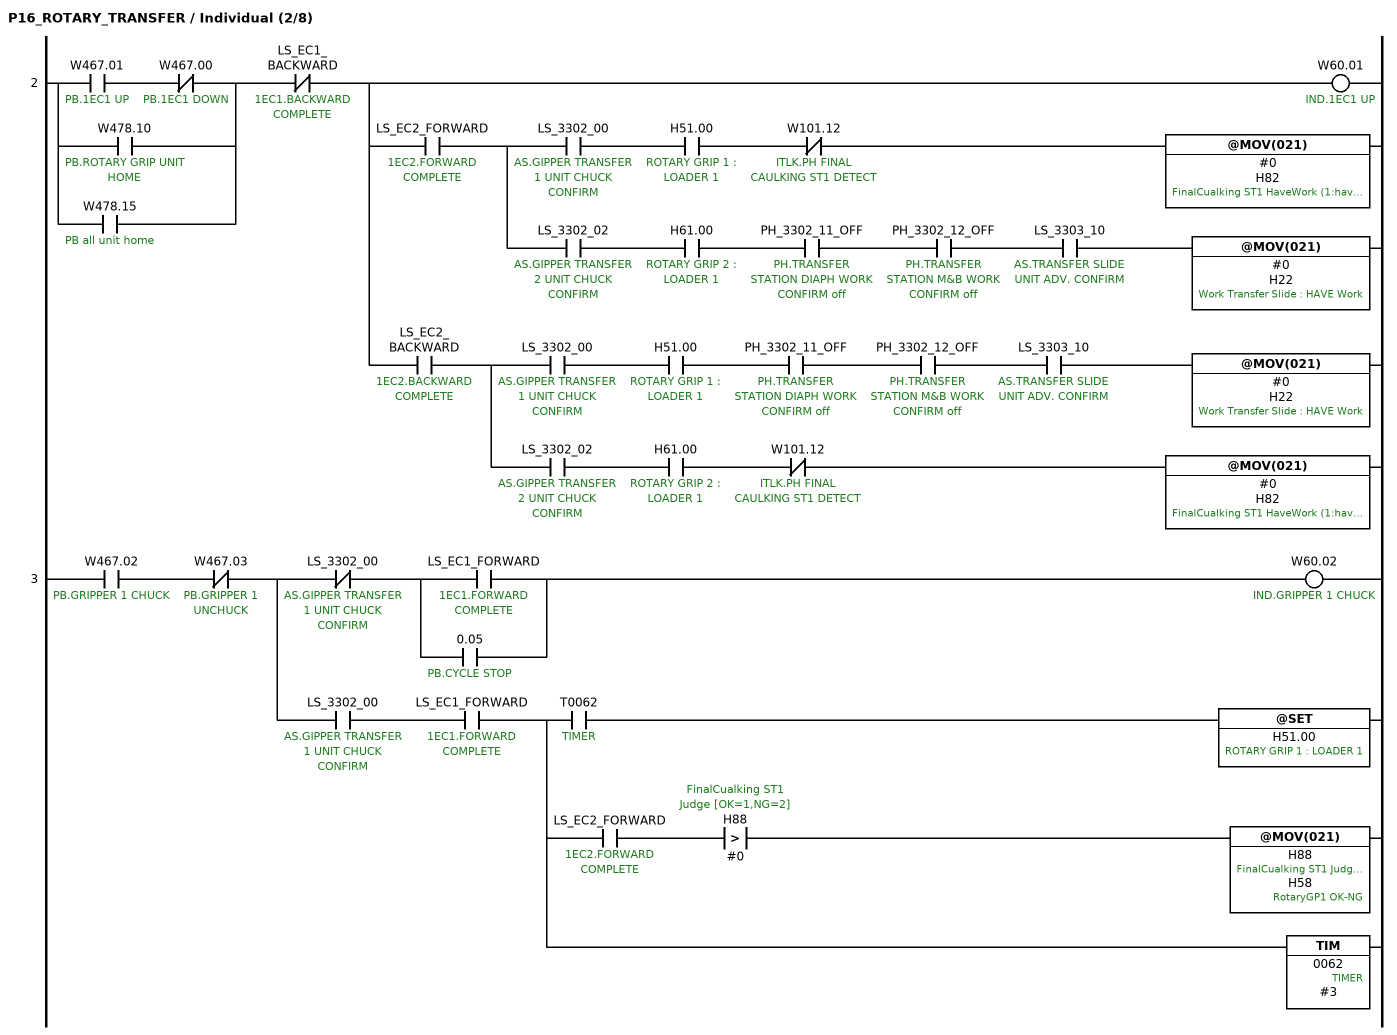
; rung 2
LD W467.01  ; PB.1EC1 UP
ANDNOT W467.00  ; PB.1EC1 DOWN
OR W478.10  ; PB.ROTARY GRIP UNIT HOME
OR W478.15  ; PB all unit home
ANDNOT LS_EC1_BACKWARD  ; 1EC1.BACKWARD COMPLETE
OUT TR0
OUT W60.01  ; IND.1EC1 UP
AND LS_EC2_FORWARD  ; 1EC2.FORWARD COMPLETE
OUT TR1
AND LS_3302_00  ; AS.GIPPER TRANSFER 1 UNIT CHUCK CONFIRM
AND H51.00  ; ROTARY GRIP 1 : LOADER 1
ANDNOT W101.12  ; ITLK.PH FINAL CAULKING ST1 DETECT
@MOV(021) #0 H82  ; FinalCualking ST1 HaveWork (1:have work 2:no work)
LD TR1
AND LS_3302_02  ; AS.GIPPER TRANSFER 2 UNIT CHUCK CONFIRM
AND H61.00  ; ROTARY GRIP 2 : LOADER 1
AND PH_3302_11_OFF  ; PH.TRANSFER STATION DIAPH WORK CONFIRM off
AND PH_3302_12_OFF  ; PH.TRANSFER STATION M&B WORK CONFIRM off
AND LS_3303_10  ; AS.TRANSFER SLIDE UNIT ADV. CONFIRM
@MOV(021) #0 H22  ; Work Transfer Slide : HAVE Work
LD TR0
AND LS_EC2_BACKWARD  ; 1EC2.BACKWARD COMPLETE
OUT TR0
AND LS_3302_00  ; AS.GIPPER TRANSFER 1 UNIT CHUCK CONFIRM
AND H51.00  ; ROTARY GRIP 1 : LOADER 1
AND PH_3302_11_OFF  ; PH.TRANSFER STATION DIAPH WORK CONFIRM off
AND PH_3302_12_OFF  ; PH.TRANSFER STATION M&B WORK CONFIRM off
AND LS_3303_10  ; AS.TRANSFER SLIDE UNIT ADV. CONFIRM
@MOV(021) #0 H22  ; Work Transfer Slide : HAVE Work
LD TR0
AND LS_3302_02  ; AS.GIPPER TRANSFER 2 UNIT CHUCK CONFIRM
AND H61.00  ; ROTARY GRIP 2 : LOADER 1
ANDNOT W101.12  ; ITLK.PH FINAL CAULKING ST1 DETECT
@MOV(021) #0 H82  ; FinalCualking ST1 HaveWork (1:have work 2:no work)
; rung 3
LD W467.02  ; PB.GRIPPER 1 CHUCK
ANDNOT W467.03  ; PB.GRIPPER 1 UNCHUCK
OUT TR0
ANDNOT LS_3302_00  ; AS.GIPPER TRANSFER 1 UNIT CHUCK CONFIRM
LD LS_EC1_FORWARD  ; 1EC1.FORWARD COMPLETE
OR 0.05  ; PB.CYCLE STOP
ANDLD
OUT W60.02  ; IND.GRIPPER 1 CHUCK
LD TR0
AND LS_3302_00  ; AS.GIPPER TRANSFER 1 UNIT CHUCK CONFIRM
AND LS_EC1_FORWARD  ; 1EC1.FORWARD COMPLETE
OUT TR0
AND T0062  ; TIMER
@SET H51.00  ; ROTARY GRIP 1 : LOADER 1
LD TR0
AND LS_EC2_FORWARD  ; 1EC2.FORWARD COMPLETE
AND>(320) H88 #0  ; FinalCualking ST1 Judge [OK=1,NG=2]
@MOV(021) H88 H58  ; FinalCualking ST1 Judge [OK=1,NG=2], RotaryGP1 OK-NG
LD TR0
TIM 0062 #3  ; TIMER

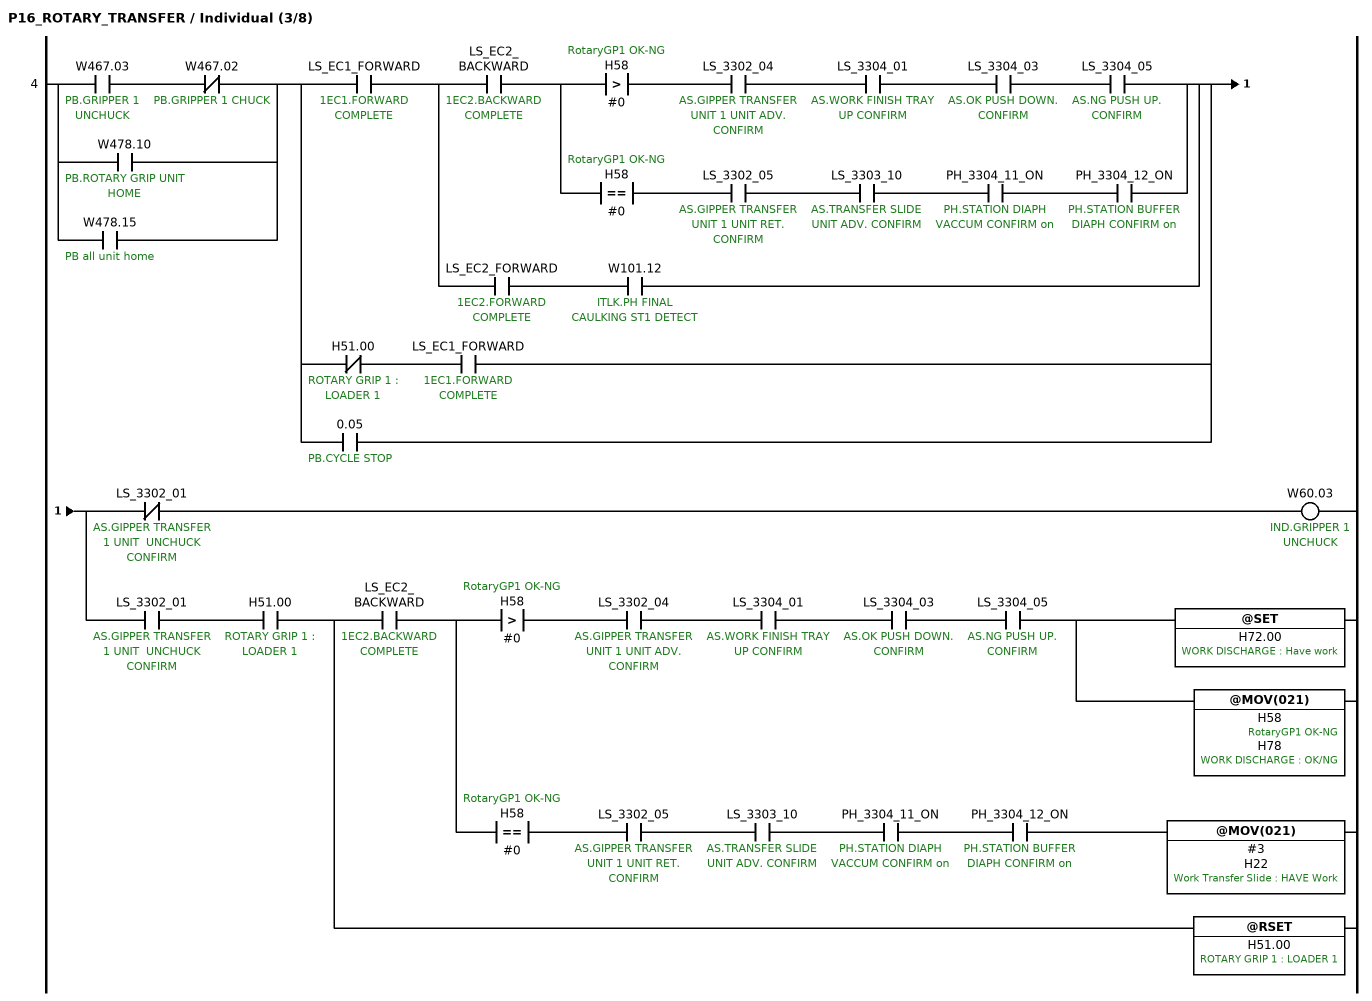
; rung 4
LD W467.03  ; PB.GRIPPER 1 UNCHUCK
ANDNOT W467.02  ; PB.GRIPPER 1 CHUCK
OR W478.10  ; PB.ROTARY GRIP UNIT HOME
OR W478.15  ; PB all unit home
LD LS_EC1_FORWARD  ; 1EC1.FORWARD COMPLETE
LD LS_EC2_BACKWARD  ; 1EC2.BACKWARD COMPLETE
LD>(320) H58 #0  ; RotaryGP1 OK-NG
AND LS_3302_04  ; AS.GIPPER TRANSFER UNIT 1 UNIT ADV. CONFIRM
AND LS_3304_01  ; AS.WORK FINISH TRAY UP CONFIRM
AND LS_3304_03  ; AS.OK PUSH DOWN. CONFIRM
AND LS_3304_05  ; AS.NG PUSH UP. CONFIRM
LD=(300) H58 #0  ; RotaryGP1 OK-NG
AND LS_3302_05  ; AS.GIPPER TRANSFER UNIT 1 UNIT RET. CONFIRM
AND LS_3303_10  ; AS.TRANSFER SLIDE UNIT ADV. CONFIRM
AND PH_3304_11_ON  ; PH.STATION DIAPH VACCUM CONFIRM on
AND PH_3304_12_ON  ; PH.STATION BUFFER DIAPH CONFIRM on
ORLD
ANDLD
LD LS_EC2_FORWARD  ; 1EC2.FORWARD COMPLETE
AND W101.12  ; ITLK.PH FINAL CAULKING ST1 DETECT
ORLD
ANDLD
LDNOT H51.00  ; ROTARY GRIP 1 : LOADER 1
AND LS_EC1_FORWARD  ; 1EC1.FORWARD COMPLETE
ORLD
OR 0.05  ; PB.CYCLE STOP
ANDLD
OUT TR0
ANDNOT LS_3302_01  ; AS.GIPPER TRANSFER 1 UNIT  UNCHUCK CONFIRM
OUT W60.03  ; IND.GRIPPER 1 UNCHUCK
LD TR0
AND LS_3302_01  ; AS.GIPPER TRANSFER 1 UNIT  UNCHUCK CONFIRM
AND H51.00  ; ROTARY GRIP 1 : LOADER 1
OUT TR0
AND LS_EC2_BACKWARD  ; 1EC2.BACKWARD COMPLETE
OUT TR1
AND>(320) H58 #0  ; RotaryGP1 OK-NG
AND LS_3302_04  ; AS.GIPPER TRANSFER UNIT 1 UNIT ADV. CONFIRM
AND LS_3304_01  ; AS.WORK FINISH TRAY UP CONFIRM
AND LS_3304_03  ; AS.OK PUSH DOWN. CONFIRM
AND LS_3304_05  ; AS.NG PUSH UP. CONFIRM
@SET H72.00  ; WORK DISCHARGE : Have work
@MOV(021) H58 H78  ; RotaryGP1 OK-NG, WORK DISCHARGE : OK/NG
LD TR1
AND=(300) H58 #0  ; RotaryGP1 OK-NG
AND LS_3302_05  ; AS.GIPPER TRANSFER UNIT 1 UNIT RET. CONFIRM
AND LS_3303_10  ; AS.TRANSFER SLIDE UNIT ADV. CONFIRM
AND PH_3304_11_ON  ; PH.STATION DIAPH VACCUM CONFIRM on
AND PH_3304_12_ON  ; PH.STATION BUFFER DIAPH CONFIRM on
@MOV(021) #3 H22  ; Work Transfer Slide : HAVE Work
LD TR0
@RSET H51.00  ; ROTARY GRIP 1 : LOADER 1

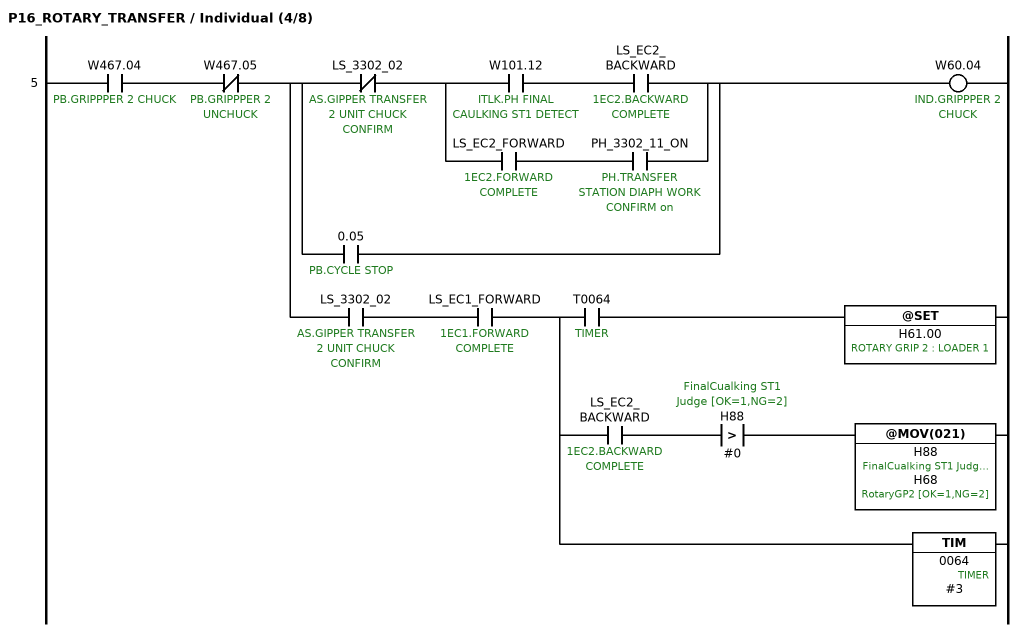
; rung 5
LD W467.04  ; PB.GRIPPPER 2 CHUCK
ANDNOT W467.05  ; PB.GRIPPPER 2 UNCHUCK
OUT TR0
LDNOT LS_3302_02  ; AS.GIPPER TRANSFER 2 UNIT CHUCK CONFIRM
LD W101.12  ; ITLK.PH FINAL CAULKING ST1 DETECT
AND LS_EC2_BACKWARD  ; 1EC2.BACKWARD COMPLETE
LD LS_EC2_FORWARD  ; 1EC2.FORWARD COMPLETE
AND PH_3302_11_ON  ; PH.TRANSFER STATION DIAPH WORK CONFIRM on
ORLD
ANDLD
OR 0.05  ; PB.CYCLE STOP
ANDLD
OUT W60.04  ; IND.GRIPPPER 2 CHUCK
LD TR0
AND LS_3302_02  ; AS.GIPPER TRANSFER 2 UNIT CHUCK CONFIRM
AND LS_EC1_FORWARD  ; 1EC1.FORWARD COMPLETE
OUT TR0
AND T0064  ; TIMER
@SET H61.00  ; ROTARY GRIP 2 : LOADER 1
LD TR0
AND LS_EC2_BACKWARD  ; 1EC2.BACKWARD COMPLETE
AND>(320) H88 #0  ; FinalCualking ST1 Judge [OK=1,NG=2]
@MOV(021) H88 H68  ; FinalCualking ST1 Judge [OK=1,NG=2], RotaryGP2 [OK=1,NG=2]
LD TR0
TIM 0064 #3  ; TIMER

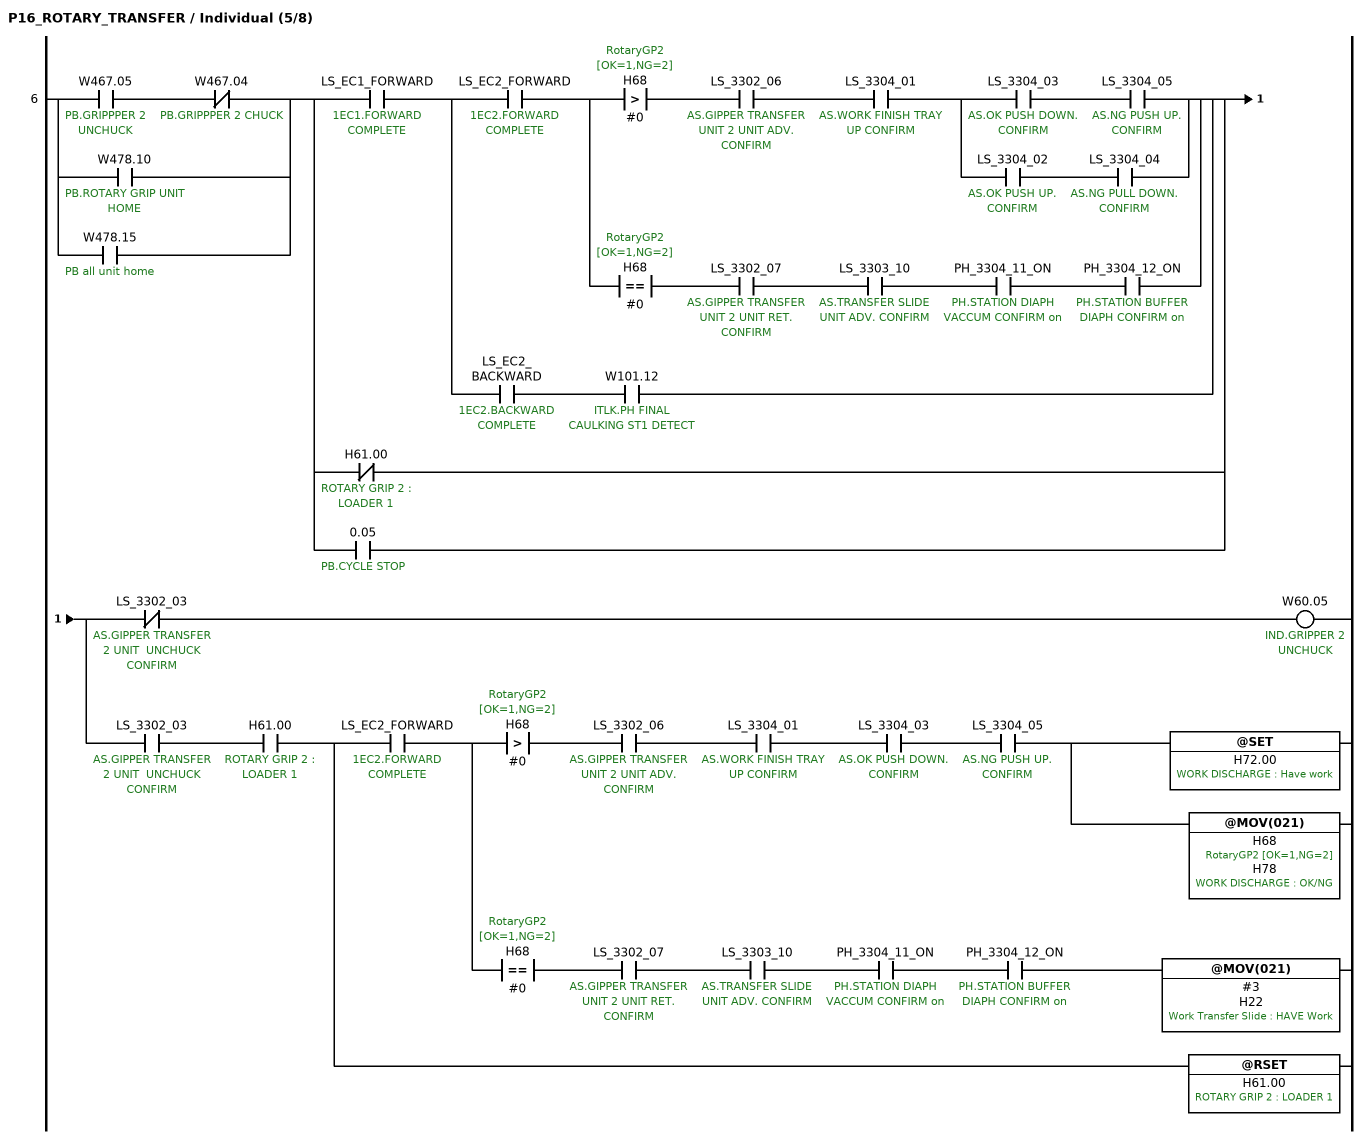
; rung 6
LD W467.05  ; PB.GRIPPPER 2 UNCHUCK
ANDNOT W467.04  ; PB.GRIPPPER 2 CHUCK
OR W478.10  ; PB.ROTARY GRIP UNIT HOME
OR W478.15  ; PB all unit home
LD LS_EC1_FORWARD  ; 1EC1.FORWARD COMPLETE
LD LS_EC2_FORWARD  ; 1EC2.FORWARD COMPLETE
LD>(320) H68 #0  ; RotaryGP2 [OK=1,NG=2]
AND LS_3302_06  ; AS.GIPPER TRANSFER UNIT 2 UNIT ADV. CONFIRM
AND LS_3304_01  ; AS.WORK FINISH TRAY UP CONFIRM
LD LS_3304_03  ; AS.OK PUSH DOWN. CONFIRM
AND LS_3304_05  ; AS.NG PUSH UP. CONFIRM
LD LS_3304_02  ; AS.OK PUSH UP. CONFIRM
AND LS_3304_04  ; AS.NG PULL DOWN. CONFIRM
ORLD
ANDLD
LD=(300) H68 #0  ; RotaryGP2 [OK=1,NG=2]
AND LS_3302_07  ; AS.GIPPER TRANSFER UNIT 2 UNIT RET. CONFIRM
AND LS_3303_10  ; AS.TRANSFER SLIDE UNIT ADV. CONFIRM
AND PH_3304_11_ON  ; PH.STATION DIAPH VACCUM CONFIRM on
AND PH_3304_12_ON  ; PH.STATION BUFFER DIAPH CONFIRM on
ORLD
ANDLD
LD LS_EC2_BACKWARD  ; 1EC2.BACKWARD COMPLETE
AND W101.12  ; ITLK.PH FINAL CAULKING ST1 DETECT
ORLD
ANDLD
ORNOT H61.00  ; ROTARY GRIP 2 : LOADER 1
OR 0.05  ; PB.CYCLE STOP
ANDLD
OUT TR0
ANDNOT LS_3302_03  ; AS.GIPPER TRANSFER 2 UNIT  UNCHUCK CONFIRM
OUT W60.05  ; IND.GRIPPER 2 UNCHUCK
LD TR0
AND LS_3302_03  ; AS.GIPPER TRANSFER 2 UNIT  UNCHUCK CONFIRM
AND H61.00  ; ROTARY GRIP 2 : LOADER 1
OUT TR0
AND LS_EC2_FORWARD  ; 1EC2.FORWARD COMPLETE
OUT TR1
AND>(320) H68 #0  ; RotaryGP2 [OK=1,NG=2]
AND LS_3302_06  ; AS.GIPPER TRANSFER UNIT 2 UNIT ADV. CONFIRM
AND LS_3304_01  ; AS.WORK FINISH TRAY UP CONFIRM
AND LS_3304_03  ; AS.OK PUSH DOWN. CONFIRM
AND LS_3304_05  ; AS.NG PUSH UP. CONFIRM
@SET H72.00  ; WORK DISCHARGE : Have work
@MOV(021) H68 H78  ; RotaryGP2 [OK=1,NG=2], WORK DISCHARGE : OK/NG
LD TR1
AND=(300) H68 #0  ; RotaryGP2 [OK=1,NG=2]
AND LS_3302_07  ; AS.GIPPER TRANSFER UNIT 2 UNIT RET. CONFIRM
AND LS_3303_10  ; AS.TRANSFER SLIDE UNIT ADV. CONFIRM
AND PH_3304_11_ON  ; PH.STATION DIAPH VACCUM CONFIRM on
AND PH_3304_12_ON  ; PH.STATION BUFFER DIAPH CONFIRM on
@MOV(021) #3 H22  ; Work Transfer Slide : HAVE Work
LD TR0
@RSET H61.00  ; ROTARY GRIP 2 : LOADER 1

